// TwinCAT 3 PLC project kittingDeca
// ProgramVersion: 3.1.4023.0
// libraries:
//   Tc2_EtherCAT, * (Beckhoff Automation GmbH)
//   Tc2_MC2, * (Beckhoff Automation GmbH)
//   Tc2_SerialCom, * (Beckhoff Automation GmbH)
//   Tc2_Standard, * (Beckhoff Automation GmbH)
//   Tc2_System, * (Beckhoff Automation GmbH)
//   Tc2_Utilities, * (Beckhoff Automation GmbH)
//   Tc3_Module, * (Beckhoff Automation GmbH)
//   VisuDialogs, * (System)
//   VisuSymbols,3.5.10.0,System
// project tree:
//   DUTs/ user_defined_structure.TcDUT
//   / GlobalTextList.TcGTLO, PlcTask.TcTTO, VISU_TASK.TcTTO, 视图管理器.TcVMO (not stored)
//   GVLs/ E_DOutputMode.TcDUT, E_State.TcDUT, ST_DIO.TcDUT, ST_IO.TcDUT, ST_IO_16.TcDUT, ST_IO_16_int.TcDUT
//   GVLs/kitting deca/axis/ AxisHMI_Ex.TcVIS, E_HomingSteps.TcDUT, FB_MotionAxis_MC.TcPOU, MC_HomeAxis.TcPOU, ST_MotionAxis_MC.TcDUT
//   GVLs/kitting deca/ DigitalInputStatus.TcDUT, FB_DigitalInput.TcPOU, FB_do.TcPOU, FB_PhotoSensor.TcPOU, Roller.TcDUT, Sensor.TcDUT, Valve.TcDUT
//   GVLs/kitting deca/measuring/ ST_byte.TcDUT, ST_IO_byte.TcDUT
//   GVLs/kitting deca/picking module/ Belt.TcDUT, Buffer.TcDUT, Inner_conveyor.TcDUT, PM_others.TcDUT, Outter_coveyor.TcDUT, Picking_Module.TcDUT, RFID.TcDUT
//   GVLs/kitting deca/replenishment module/ arLiftAxis.TcDUT, Infeed.TcDUT, Lift.TcDUT, Outfeed.TcDUT, Replenishment_Module.TcDUT
//   POUs/ E_RemIndex.TcDUT, FB_axisCtrl.TcPOU, FB_remAxisMapping.TcPOU, FB_pmAxisMapping.TcPOU, FB_remIOmapping.TcPOU, FB_rmIOmapping.TcPOU, G_HMI.TcGVL, GVL.TcGVL, G_IO.TcGVL, MAIN.TcPOU, ST_axisCtrl.TcDUT, ST_Color.TcDUT
//   VISUs/ OtherList.TcVIS, visu_PM.TcVIS, visu_ReM.TcVIS, visu_MLC.TcVIS, visu_main.TcVIS, ReMList.TcVIS, PMList.TcVIS, v_byte.TcVIS, v_IO_ReM.TcVIS, v_rem_0.TcVIS, v_pm_0.TcVIS, v_rem_1.TcVIS
// real-time tasks:
//   TASK PlcTask: cycle T#1ms, priority 20, ADS port 350
//   TASK VISU_TASK: cycle T#200000us, priority 30, ADS port 351
// motion (NC):
//   TASK NC-Task 1 SAF: cycle T#2ms, priority 4, ADS port 501
//   TASK NC-Task 1 SVB: cycle T#10ms, priority 8, ADS port 511
//   AXIS rem0_Lift0 (id 4)
//     Dynamic: Acceleration=15000, Deceleration=15000, Jerk=150000
//     Velo: Maximum=3000
//     OtherSettings: AllowMotionCmdToSlave=true
//     encoder EncType=19
//       EncPara: ScaleFactorNumerator=5, ScaleFactorDenominator=262144, Inverse=true, MaxCount=#xffffffff
//         Inc: RefSoftSyncMask=#x00040000
//     drive DrvType=16
//       DrvPara: Inverse=true, MaxCount=#xffffffff, DriveControlDWord=#x00020100
//         Analog: VeloReferenz=500, TorqueSetpointScale=10, ScaleFactorActTorque=0.1
//         TimeComp: TaskDelayCycles=1
//     controller CtrType=1
//       CtrPara: PriorControlFactor=1
//         PosDiffControl: Range=30
//         Observer: BandWidth=20
//   AXIS rem0_Lift1 (id 5)
//     Dynamic: Acceleration=15000, Deceleration=15000, Jerk=150000
//     Velo: Maximum=3000
//     OtherSettings: AllowMotionCmdToSlave=true
//     encoder EncType=19
//       EncPara: ScaleFactorNumerator=5, ScaleFactorDenominator=262144, Inverse=true, MaxCount=#xffffffff
//         Inc: RefSoftSyncMask=#x00040000
//     drive DrvType=16
//       DrvPara: Inverse=true, MaxCount=#xffffffff, DriveControlDWord=#x00020100
//         Analog: VeloReferenz=500, TorqueSetpointScale=10, ScaleFactorActTorque=0.1
//         TimeComp: TaskDelayCycles=1
//     controller CtrType=1
//       CtrPara: PriorControlFactor=1
//         PosDiffControl: Range=30
//         Observer: BandWidth=20
//   AXIS rem1_Lift0 (id 1)
//     Dynamic: Acceleration=15000, Deceleration=15000, Jerk=150000
//     Velo: Maximum=3000
//     OtherSettings: AllowMotionCmdToSlave=true
//     encoder EncType=1
//       EncPara: ScaleFactorNumerator=5, ScaleFactorDenominator=262144, Inverse=true
//         Inc: RefSoftSyncMask=#x00040000
//     drive DrvType=5
//       DrvPara: Inverse=true
//         Analog: VeloReferenz=500, TorqueSetpointScale=10, ScaleFactorActTorque=0.1
//         TimeComp: TaskDelayCycles=1
//     controller CtrType=1
//       CtrPara: PriorControlFactor=1
//         PosDiffControl: Range=30
//         Observer: BandWidth=20
//   AXIS rem1_Lift1 (id 2)
//     Dynamic: Acceleration=15000, Deceleration=15000, Jerk=150000
//     Velo: Maximum=3000
//     OtherSettings: AllowMotionCmdToSlave=true
//     encoder EncType=1
//       EncPara: ScaleFactorNumerator=5, ScaleFactorDenominator=262144, Inverse=true
//         Inc: RefSoftSyncMask=#x00040000
//     drive DrvType=5
//       DrvPara: Inverse=true
//         Analog: VeloReferenz=500, TorqueSetpointScale=10, ScaleFactorActTorque=0.1
//         TimeComp: TaskDelayCycles=1
//     controller CtrType=1
//       CtrPara: PriorControlFactor=1
//         PosDiffControl: Range=30
//         Observer: BandWidth=20
// I/O:
//   DEVICE LB Test (EtherCAT) (disabled), AmsNetId 172.18.236.248.8.1
//     Box 19 (GL20-RTU-ECT) [GL20-RTU-ECT_1.3.5.0]
//       modules: Module 1 (GL20-1600END), Module 2 (GL20-0016ETP)
//     Drive 20 (InoMD800) [MD800_ECAT_9Axis_V0.19]
//   DEVICE ReM test, AmsNetId 192.168.11.159.7.2
//     Box 8 (GL20-RTU-ECT) [GL20-RTU-ECT_1.3.5.0]
//       modules: Module 1 (GL20-1600END), Module 2 (GL20-1600END), Module 3 (GL20-1600END), Module 4 (GL20-1600END), Module 5 (GL20-0016ETP), Module 6 (GL20-0016ETP)
//     rem0_lift0(InoSV630N) [SV630_1Axis_03713]
//     rem0_lift1(InoSV630N) [SV630_1Axis_03713]
//     Box 22 (C2S-EC) [C2S-EC]
//       modules: Module 1 (C2S-EC-24B)
//     Box 25 (6076924) [SIG350-0006AP100] (disabled)
//       modules: Module 1 (IOL_32/32_I/O-Bytes), Module 2 (IOL_32/32_I/O-Bytes), Module 3 (Digital_IN), Module 4 (Digital_IN), Module 5 (Digital_IN), Module 6 (Digital_IN), Module 7 (Digital_IN), Module 8 (Digital_IN)
// variable links:
//   NC-Task 1 SAF/Axes/rem0_Lift0 <-> ReM test/rem0_lift0(InoSV630N)
//     Drive/Inputs/In/nDataIn1 <-> Inputs/Following error actual value
//     Drive/Inputs/In/nDataIn3[0] <-> Inputs/Torque actual value
//     Drive/Inputs/In/nDcOutputTime <-> InfoData/DcOutputShift
//     Drive/Inputs/In/nState1 <-> Inputs/Statusword
//     Drive/Inputs/In/nState2 <-> Inputs/Statusword @bit 8
//     Drive/Inputs/In/nState4 @bit 1 <-> WcState/InputToggle
//     Drive/Inputs/In/nState4 <-> WcState/WcState
//     Drive/Outputs/Out/nCtrl1 <-> Outputs/Controlword
//     Drive/Outputs/Out/nCtrl2 <-> Outputs/Controlword @bit 8
//     Drive/Outputs/Out/nDataOut1 <-> Outputs/Target position
//     Enc/Inputs/In/nDataIn1 <-> Inputs/Position actual value
//     Enc/Inputs/In/nDataIn3 <-> Inputs/Touch probe pos1 pos value
//     Enc/Inputs/In/nDataIn5 <-> Inputs/Touch probe pos2 pos value
//     Enc/Inputs/In/nDcInputTime <-> InfoData/DcInputShift
//     Enc/Inputs/In/nState4 @bit 1 <-> WcState/InputToggle
//     Enc/Inputs/In/nState4 <-> WcState/WcState
//     Enc/Inputs/In/nState5 <-> Inputs/Touch probe status
//     Enc/Inputs/In/nState6 <-> Inputs/Touch probe status @bit 8
//     Enc/Outputs/Out/nCtrl5 <-> Outputs/Touch probe function
//     Enc/Outputs/Out/nCtrl6 <-> Outputs/Touch probe function @bit 8
//   NC-Task 1 SAF/Axes/rem0_Lift1 <-> ReM test/rem0_lift1(InoSV630N)
//     Drive/Inputs/In/nDataIn1 <-> Inputs/Following error actual value
//     Drive/Inputs/In/nDataIn3[0] <-> Inputs/Torque actual value
//     Drive/Inputs/In/nDcOutputTime <-> InfoData/DcOutputShift
//     Drive/Inputs/In/nState1 <-> Inputs/Statusword
//     Drive/Inputs/In/nState2 <-> Inputs/Statusword @bit 8
//     Drive/Inputs/In/nState4 @bit 1 <-> WcState/InputToggle
//     Drive/Inputs/In/nState4 <-> WcState/WcState
//     Drive/Outputs/Out/nCtrl1 <-> Outputs/Controlword
//     Drive/Outputs/Out/nCtrl2 <-> Outputs/Controlword @bit 8
//     Drive/Outputs/Out/nDataOut1 <-> Outputs/Target position
//     Enc/Inputs/In/nDataIn1 <-> Inputs/Position actual value
//     Enc/Inputs/In/nDataIn3 <-> Inputs/Touch probe pos1 pos value
//     Enc/Inputs/In/nDataIn5 <-> Inputs/Touch probe pos2 pos value
//     Enc/Inputs/In/nDcInputTime <-> InfoData/DcInputShift
//     Enc/Inputs/In/nState4 @bit 1 <-> WcState/InputToggle
//     Enc/Inputs/In/nState4 <-> WcState/WcState
//     Enc/Inputs/In/nState5 <-> Inputs/Touch probe status
//     Enc/Inputs/In/nState6 <-> Inputs/Touch probe status @bit 8
//     Enc/Outputs/Out/nCtrl5 <-> Outputs/Touch probe function
//     Enc/Outputs/Out/nCtrl6 <-> Outputs/Touch probe function @bit 8
//   kittingDeca/kittingDeca Instance <-> NC-Task 1 SAF/Axes/rem0_Lift0
//     PlcTask Inputs/GVL.rem[0].lift[0].AxisRef.NcToPlc <-> Outputs/ToPlc
//     PlcTask Outputs/GVL.rem[0].lift[0].AxisRef.PlcToNc <-> Inputs/FromPlc
//   kittingDeca/kittingDeca Instance <-> NC-Task 1 SAF/Axes/rem0_Lift1
//     PlcTask Inputs/GVL.rem[0].lift[1].AxisRef.NcToPlc <-> Outputs/ToPlc
//     PlcTask Outputs/GVL.rem[0].lift[1].AxisRef.PlcToNc <-> Inputs/FromPlc

CONFIGURATION kittingDeca
    RESOURCE PLC ON TwinCAT3
        TASK PlcTask(INTERVAL := T#1ms, PRIORITY := 20);
        TASK VISU_TASK(INTERVAL := T#200000us, PRIORITY := 30);
        PROGRAM MAIN WITH PlcTask : MAIN;
        PROGRAM VisuElems_Visu_Prg WITH VISU_TASK : VisuElems.Visu_Prg;
    END_RESOURCE
END_CONFIGURATION

// ---- DUTs/user_defined_structure.TcDUT
{attribute 'pack_mode' := '1'}
TYPE user_defined_structure :
STRUCT
	a:BOOL;
	b:INT;
	c:STRING;
	d:REAL;
END_STRUCT
END_TYPE

// ---- GVLs/E_DOutputMode.TcDUT
{attribute 'qualified_only'}
{attribute 'strict'}
TYPE E_DOutputMode :
(
	AutoPLC 	:= 0,
	ManualHMI	:= 1
);
END_TYPE

// ---- GVLs/E_State.TcDUT
{attribute 'qualified_only'}
{attribute 'strict'}
TYPE E_State :
(
	DISABLE		:= 0,
	READY 		:= 1,
	WARNING		:= 2,
	ERROR		:= 3
	
);
END_TYPE

// ---- GVLs/kitting deca/axis/E_HomingSteps.TcDUT
TYPE E_HomingSteps :
(
	IDLE 				:= 0,
	INIT				:= 5,
	READ_AND_SAVE_PARAM	:= 10,
	DISABLE_SOFT_LIM	:= 15,
	ENABLE_JOG			:= 20,
	HOMING				:= 25,
	SET_POSITION		:= 30,
	START					:=	40,
	CHECK					:=	45,
	JOG_FW					:=	100,
	JOG_BW_DOG				:=	105,
	FW_DOG_OFF				:=	110,
	BW_DOG_ON				:=	115,
	
	JOG_BW					:=	130,
	JOG_FW_DOG				:=	135,
	BW_DOG_OFF				:=	140,
	FW_DOG_ON				:=	145,
	MCHOME					:=	150,
	WAIT					:=	160,
	DONE				:= 800,
	ERROR				:= 900
);
END_TYPE

// ---- GVLs/kitting deca/axis/ST_MotionAxis_MC.TcDUT
TYPE ST_MotionAxis_MC :
STRUCT
	rVelocity						: 	LREAL   						;
	rVelocity2						: 	LREAL   						;
	rMaxVelocity					:	LREAL							;	
	rAcceleration					:	LREAL							;
	rMaxAcceleration				:	LREAL							;
	rDeceleration					:	LREAL   						;
	rMaxDeceleration				:	LREAL							;
	rJerk							:	LREAL							;
	rMaxJerk						:	LREAL							;
	rPosition						:	LREAL							;
	rSetPosDistance					:	LREAL							;
	rSetPos							: 	LREAL							;	
	rDistance						:   LREAL							;
	rDistance2						:   LREAL							;	
	
	rActualPosSet					:	LREAL							;//ADD BY EVAN 
	rVelocitySet					: 	LREAL   						;//ADD BY EVAN 	
	xHoming							:	BOOL							;//ADD BY EVAN 
	
	rMaxDistance					:	LREAL							;
	bLimit							:   BOOL							;
	bNegLim							:   BOOL							;
	bPosLim							:	BOOL							;
	bNegSen							:   BOOL							;
	bPosSen							:	BOOL							;
	bPositionSensor					:	BOOL							;
	rHomePos						:	LREAL							;
	rActualPos						:	LREAL							;
	PosDiff							:	LREAL							;
	rActualCurr						:	LREAL							;
	axisDirection					:	MC_Direction					;
	
	rVeloPers						: 	LREAL							;
	rAccPers						: 	LREAL							;   
	rDecPers						: 	LREAL							;                                             					
	SetHomePos						: 	LREAL							;
	HomeVelo						: 	LREAL							;
	PosDiffTarget					: 	LREAL							;
	rFirstpos						: 	LREAL							;
	iAxisID							:	INT								;
	xhsHomingStart					: 	BOOL							;
	xHomingDone						: 	BOOL							;
	xForceControlStart				: 	BOOL							;
	xFoceControlDone				:	BOOL							;	
	xMoveABSDone					: 	BOOL							;
	xMoveRelDone					:	BOOL							;
	bInCouple						:	BOOL							;//Flag Axis is coupled 
    xMuteAxisErrorMessages			:	BOOL							;                                         					
	//Visible/Hide HMI interfaces                   					
	bHomeButtonShow					:	BOOL							; 
	bNegSensorShow					:	BOOL							; 
	bPosSensorShow					:	BOOL							;
	bBacklashShow					:	BOOL							;
	bUnitDegShow					:	BOOL							;
    bJerkShow						:	BOOL							; 
	bStopButtonShow					:	BOOL							; 
	   
	
	bMoveAbsHMI						:	BOOL;
	rVelocityHMI 					: 	LREAL;
	rActualPosHMI					:	LREAL							;//ADD BY EVAN
	bMChomingEnable					:	BOOL							;                                         				
	// backlash compensation                        	
	rBacklashvalue					:	LREAL							;
	xbacklashEnable					:	BOOL							;                        		                					
	bdirFW							:	BOOL							;// on hard stop homing , define the direction of rotation
	
	ModOp					 		: 	SINT							;// Axis operation mode (8 )

//	==============================	Beckhoff Tc2_MC2 library(motion)	==================================
	mcPower 						: 	MC_Power					    ;(*	Axis power, enable/disable																			*)
	mcAxisStates					:	MC_AxisStates					;(*	Driver Feedback, curr motor stage 																	*)
	mcHalt							: 	MC_Halt							;(*	Stops an axis with a defined braking ramp															*)
	mcHome							: 	MC_Home							;(*	Axis homing scenario and execution																	*)
	mcJog							: 	MC_Jog							;(*	Axis Joging BW/FW																					*)	
	mcMoveAbsolute					: 	MC_MoveAbsolute					;(*	Axis GoTo Absolute position																			*)	
	mcMoveRelative					: 	MC_MoveRelative					;(*	Axis GoTo Step by SetPos +/- actual position														*)
	mcMoveVelocity					: 	MC_MoveVelocity					;(*	Axis GoTo with constant velocity														*)
	mcReadStatus					: 	MC_ReadStatus					;(*	Read Axis statuses from driver																		*)
	mcReset							: 	MC_Reset						;(*	Reset Driver																						*)
	mcStop							: 	MC_Stop							;(*	Stop Driver																							*)
	mcReadActualPosition			:	MC_ReadActualPosition			;(*	Read the current axis position																		*)
	mcSetpoint						: 	MC_SetPosition					;(*	Sets the current axis position to a parameterizable value											*)
	mcWriteBoolParameter			: 	MC_WriteBoolParameter			;(*	Write bool param to driver																			*)
	mcReadBoolParameter				:	MC_ReadBoolParameter			;(*	Read bool param from driver																			*)
	mcAxisParameter					:   MC_AxisParameter				;(*	Data type is used in conjunction with function blocks for reading and writing of axis parameters	*)
	CoeWrt							:	FB_EcCoESdoWrite;											
	
//	======================================================================================================	

//
	iSdoWrite	:INT; //6:clear encoder
	sNetID : STRING;
	nSlaveAddr	:UINT;
	nSubIndex	: BYTE;
	nIndex	: WORD;
	
	iCoeWrt	: INT;

END_STRUCT
END_TYPE

// ---- GVLs/kitting deca/DigitalInputStatus.TcDUT

{attribute 'qualified_only'}
{attribute 'strict'}
TYPE DigitalInputStatus:
(
        LOW := 0,
        HIGH := 1
);
END_TYPE

// ---- GVLs/kitting deca/measuring/ST_byte.TcDUT
TYPE ST_byte :
STRUCT
	arByte				: ARRAY[1..32] OF ST_IO_byte; 	// struct of digital Imputs for use in program and hmi 
END_STRUCT
END_TYPE

// ---- GVLs/kitting deca/measuring/ST_IO_byte.TcDUT
TYPE ST_IO_byte : // struct of digital IO for use in program and hmi 
STRUCT
	Ch : ARRAY[0..7] OF BOOL ;

END_STRUCT
END_TYPE

// ---- GVLs/kitting deca/picking module/Belt.TcDUT
TYPE Belt :
STRUCT
	cmd	: INT;
	freq	: INT;
END_STRUCT
END_TYPE

// ---- GVLs/kitting deca/picking module/Buffer.TcDUT
TYPE Buffer :
STRUCT
	mcAxis 					: FB_MotionAxis_MC;
	st_mcAxis 				: ST_MotionAxis_MC;
	AxisRef					: AXIS_REF;
	axis_sensor	: BOOL;
	power_axis	: BOOL;
	contractor_axis	: BOOL;
	surfae_slot_0	: BOOL;
	surfae_slot_1	: BOOL;
	surfae_slot_2	: BOOL;
	above_fixture_light_curtain	: BOOL;
	lamp_button	: BOOL;
	button	: BOOL;
	locked	: BOOL;
	magnet	: BOOL;
	magnet_locked	: BOOL;
END_STRUCT
END_TYPE

// ---- GVLs/kitting deca/picking module/Inner_conveyor.TcDUT
TYPE Inner_conveyor :
STRUCT
	belt	: ARRAY[0..2] OF Belt;
	valve	: ARRAY[0..2] OF Valve;
	rfid	: ARRAY[0..1] OF RFID;
END_STRUCT
END_TYPE

// ---- GVLs/kitting deca/picking module/PM_others.TcDUT
TYPE PM_others :
STRUCT
	power_inConv	:BOOL;
	contactor_inConv	: BOOL;
	power_outConv	:BOOL;
	contactor_outConv	: BOOL;	
	measuring_light_curtain_a	: ARRAY[0..16] OF BYTE;
	measuring_light_curtain_b	: ARRAY[0..16] OF BYTE;
END_STRUCT
END_TYPE

// ---- GVLs/kitting deca/picking module/Outter_coveyor.TcDUT
TYPE Outter_coveyor :
STRUCT
	belt	: ARRAY[0..1] OF Belt;
	valve	: ARRAY[0..1] OF Valve;
	photo_sensor	: ARRAY[0..1] OF BOOL;	
END_STRUCT
END_TYPE

// ---- GVLs/kitting deca/picking module/Picking_Module.TcDUT
TYPE Picking_Module :
STRUCT
	buffer : ARRAY[0..1]OF Buffer;	
	inConv : Inner_conveyor;
	outConv : Outter_coveyor;
	power_robot			: BOOL;
	contactor_robot		: BOOL;
	power_inConv		: BOOL;
	contactor_inConv	: BOOL;
	power_outConv		: BOOL;
	contactor_outConv	: BOOL;	
	
END_STRUCT
END_TYPE

// ---- GVLs/kitting deca/picking module/RFID.TcDUT
TYPE RFID :
STRUCT
END_STRUCT
END_TYPE

// ---- GVLs/kitting deca/replenishment module/arLiftAxis.TcDUT
TYPE arLiftAxis :
STRUCT
	lift : ARRAY[0..1] OF FB_remAxisMapping;
END_STRUCT
END_TYPE

// ---- GVLs/kitting deca/replenishment module/Infeed.TcDUT
TYPE Infeed :
STRUCT
	roller : Roller;
	valve_stopper : Valve;
	photo_sensor :ARRAY[0..1]OF FB_PhotoSensor;
END_STRUCT
END_TYPE

// ---- GVLs/kitting deca/replenishment module/Lift.TcDUT
TYPE Lift :
STRUCT
	roller : Roller;
	power_axis	: BOOL;
	contactor_axis : BOOL;	
	mcAxis 					: FB_MotionAxis_MC;
	st_mcAxis 				: ST_MotionAxis_MC;
	AxisRef					: AXIS_REF;
	valve_perturbation : ARRAY [0..3] OF Valve;
	valve_clamp	:Valve;
	photo_sensor :ARRAY[0..1]OF FB_PhotoSensor;
	limit_sensor : ARRAY[0..2]OF BOOL;

END_STRUCT
END_TYPE

// ---- GVLs/kitting deca/replenishment module/Outfeed.TcDUT
TYPE Outfeed :
STRUCT
	roller : Roller;
	photo_sensor :ARRAY[0..1]OF FB_PhotoSensor;
END_STRUCT
END_TYPE

// ---- GVLs/kitting deca/replenishment module/Replenishment_Module.TcDUT
TYPE Replenishment_Module :
STRUCT
	infeed : ARRAY[0..1]OF Infeed;
	outfeed : ARRAY[0..1]OF Outfeed;
	lift : ARRAY[0..1]OF Lift;
END_STRUCT
END_TYPE

// ---- GVLs/kitting deca/Roller.TcDUT
TYPE Roller :
STRUCT
	Power  		: BOOL;
	forward  	: BOOL; 
	backward	: BOOL;
	err 		: BOOL;
END_STRUCT
END_TYPE

// ---- GVLs/kitting deca/Sensor.TcDUT
TYPE Sensor :
STRUCT
	
END_STRUCT
END_TYPE

// ---- GVLs/kitting deca/Valve.TcDUT
TYPE Valve :
STRUCT
	extend 		 : BOOL;
	retract		 : BOOL;
	extended 	 : BOOL;
	retracted 	 : BOOL;	
END_STRUCT
END_TYPE

// ---- GVLs/ST_DIO.TcDUT
TYPE ST_DIO :
STRUCT
	arstDI				: ARRAY[0..DiMouduleMAX] OF ST_IO_16_int; 	// struct of digital Imputs for use in program and hmi 
	arstDO				: ARRAY[0..DOMODULEMAX] OF ST_IO_16_int;	// struct of digital Outputs for use in program and hmi 
	eDOutputMode		: E_DOutputMode 					;	// Switch for change sourse of DO (0 from plc, 1 from HMI)
END_STRUCT
END_TYPE

// ---- GVLs/ST_IO.TcDUT
TYPE ST_IO :
STRUCT
	sName			: STRING		;
	iState			: E_State		;
	xState			: REFERENCE TO BOOL 			;
	xStateHMI		: BOOL 			;
	xInvisible		: BOOL			;
	
END_STRUCT
END_TYPE

// ---- GVLs/ST_IO_16.TcDUT
TYPE ST_IO_16: 
STRUCT
	Ch : ARRAY[0..15] OF BOOL  ; 
END_STRUCT
END_TYPE

// ---- GVLs/ST_IO_16_int.TcDUT
TYPE ST_IO_16_int : // struct of digital IO for use in program and hmi 
STRUCT
	Ch : ARRAY[0..15] OF ST_IO ;

END_STRUCT
END_TYPE

// ---- POUs/E_RemIndex.TcDUT
{attribute 'qualified_only'}
{attribute 'strict'}
TYPE E_RemIndex :
(
	REM0		:= 0,
	REM1 		:= 1,
	REM2		:= 2,
	REM3		:= 3,
	REM4		:= 4,
	REM5 		:= 5,
	REM6		:= 6,
	REM7		:= 7,
	REM8		:= 8,
	REM9 		:= 9
);
END_TYPE

// ---- POUs/ST_axisCtrl.TcDUT
TYPE ST_axisCtrl :
STRUCT
	iStatus	: INT;
	iCmd	: INT;
	iSpeed	: INT;
	rPosition	: LREAL;
	sMsg	: STRING;
END_STRUCT
END_TYPE

// ---- POUs/ST_Color.TcDUT
TYPE ST_Color :
STRUCT
	RED			: DWORD	:= 16#FFFF0000;
	YELLOW		: DWORD	:= 16#FFFFFF00;
	GREEN		: DWORD	:= 16#FF00FF00;
	GREY		: DWORD	:= 16#FFBEBEBE;
	WHITE		: DWORD	:= 16#FFFFFFFF;
	BLACK		: DWORD	:= 16#FF000000;
	BLUE		: DWORD	:= 16#FF0000FF;
END_STRUCT
END_TYPE

// ---- POUs/G_HMI.TcGVL
{attribute 'qualified_only'}
VAR_GLOBAL
	iMainFrame : INT;
	iReM: INT;
	iPM	: INT;
END_VAR

// ---- POUs/GVL.TcGVL
{attribute 'qualified_only'}
VAR_GLOBAL CONSTANT

END_VAR
VAR_GLOBAL

	
	
	rem : ARRAY[0..9] OF Replenishment_Module;
	pm	: ARRAY[0..9] OF Picking_Module;
	pmOthers	:ARRAY[0..4] OF PM_others;
	
	

	
    stByte : REFERENCE TO ST_byte;
	ibyteNum			:ARRAY[1..32] OF  INT ;
	stMeasuringLC : ST_byte;
	byteLC AT%I*:ARRAY [1..32] OF BYTE;
	rfidIn AT%I*:ARRAY [0..31] OF BYTE;
	rfidOut AT%Q*:ARRAY [0..31] OF BYTE;
	arIn	: ARRAY[0..3] OF ST_IO_byte;
	arOut	: ARRAY[0..3] OF ST_IO_byte;
	n: INT;
	
	fb_remIOmapping	: ARRAY[0..9] OF FB_remIOmapping;
	fb_remAxisMapping	: ARRAY[0..19] OF FB_remAxisMapping;
	stAxisCtrl_Lift	: ARRAY[0..19]OF ST_axisCtrl;
	fbAxisCtrl_Lift	: ARRAY [0..19] OF FB_axisCtrl;

	fb_rmIOmapping	: ARRAY[0..4] OF FB_rmIOmapping;
	fb_pmAxisMapping	: ARRAY[0..19] OF FB_pmAxisMapping;
	stAxisCtrl_Buffer	: ARRAY[0..19]OF ST_axisCtrl;
	fbAxisCtrl_Buffer	: ARRAY [0..19] OF FB_axisCtrl;
	

	
END_VAR

// ---- POUs/G_IO.TcGVL
{attribute 'global_init_slot' := '40600'}
VAR_GLOBAL CONSTANT
	{attribute 'global_init_slot'}
	DiMouduleMAX 			:	INT	:=	100;
	{attribute 'global_init_slot'}
	DOMODULEMAX 			:	INT	:=	100;
END_VAR

VAR_GLOBAL
	{attribute 'TcContextName':='PlcTask1'}
	arDI	AT%I*		: ARRAY[0..DiMouduleMAX ] OF ST_IO_16;		//  links to Digital input  Modules 
	{attribute 'TcContextName':='PlcTask1'}
	arDO	AT%Q*		: ARRAY[0..DOMODULEMAX ] OF ST_IO_16;		//  links to Digital output Modules

	iDiMouduleMAX		: INT := 100 							; 		//Number of DI module 
	iDOModuleMax		: INT := 100 							; 		//Number of DO module 


	stDIO				: ST_DIO 							;		// struct DIO for use in plc program
		
	{attribute 'TcContextName':='PlcTask1'}
   	

END_VAR

// ---- POUs/MAIN.TcPOU
PROGRAM MAIN
VAR
	test_bool:BOOL;
	test_int:INT;
	test_real:REAL;
	test_string:STRING;
	test_arr_int:ARRAY[1..10] OF INT;
	test_word:WORD;
	test_arr_bool:ARRAY[1..3] OF BOOL;
	test_structure:user_defined_structure;
	test_arr_string:ARRAY[1..3] OF STRING;
	
	fb_Time : FB_LocalSystemTime;

	byte1 : BYTE;
	string1 :STRING;

	
END_VAR

fb_Time(bEnable := TRUE); 

M_mappingIO();
M_measuringLC();
M_rfid();
runEveryCycle();
M_ReM();

METHOD M_mappingIO 
VAR_INPUT
END_VAR
GVL.fb_remIOmapping[0](iReM:= 0);
GVL.fb_remIOmapping[1](iReM:= 1);
GVL.fb_remIOmapping[2](iReM:= 2);
GVL.fb_remIOmapping[3](iReM:= 3);
GVL.fb_remIOmapping[4](iReM:= 4);
GVL.fb_remIOmapping[5](iReM:= 5);
GVL.fb_remIOmapping[6](iReM:= 6);
GVL.fb_remIOmapping[7](iReM:= 7);
GVL.fb_remIOmapping[8](iReM:= 8);
GVL.fb_remIOmapping[9](iReM:= 9);
GVL.fb_remAxisMapping[0](iReM :=0,iLift:=0,nSlaveAddr:=1002);
GVL.fb_remAxisMapping[1](iReM :=0,iLift:=1,nSlaveAddr:=1003);
GVL.fb_remAxisMapping[2](iReM :=1,iLift:=0,nSlaveAddr:=1006);
GVL.fb_remAxisMapping[3](iReM :=1,iLift:=1,nSlaveAddr:=1007);

GVL.fbAxisCtrl_Lift[0](stAxisCtrl:=GVL.stAxisCtrl_Lift[0],IN_OUT:=GVL.rem[0].lift[0].st_mcAxis);
GVL.fbAxisCtrl_Lift[1](stAxisCtrl:=GVL.stAxisCtrl_Lift[1],IN_OUT:=GVL.rem[0].lift[1].st_mcAxis);
GVL.fbAxisCtrl_Lift[2](stAxisCtrl:=GVL.stAxisCtrl_Lift[2],IN_OUT:=GVL.rem[1].lift[0].st_mcAxis);
GVL.fbAxisCtrl_Lift[3](stAxisCtrl:=GVL.stAxisCtrl_Lift[3],IN_OUT:=GVL.rem[1].lift[1].st_mcAxis);


GVL.fb_rmIOmapping[0](iRm:= 0);
GVL.fb_rmIOmapping[0](iRm:= 1);
GVL.fb_rmIOmapping[0](iRm:= 2);
GVL.fb_rmIOmapping[0](iRm:= 3);
GVL.fb_rmIOmapping[0](iRm:= 4);
GVL.fb_pmAxisMapping[0](iPM :=0,iBuffer:=0,nSlaveAddr:=2002);
GVL.fb_pmAxisMapping[1](iPM :=0,iBuffer:=1,nSlaveAddr:=2003);
GVL.fb_pmAxisMapping[2](iPM :=1,iBuffer:=0,nSlaveAddr:=2006);
GVL.fb_pmAxisMapping[3](iPM :=1,iBuffer:=1,nSlaveAddr:=2007);
GVL.fbAxisCtrl_Buffer[0](stAxisCtrl:=GVL.stAxisCtrl_Buffer[0],IN_OUT:=GVL.pm[0].buffer[0].st_mcAxis);
GVL.fbAxisCtrl_Buffer[1](stAxisCtrl:=GVL.stAxisCtrl_Buffer[1],IN_OUT:=GVL.pm[0].buffer[1].st_mcAxis);
GVL.fbAxisCtrl_Buffer[2](stAxisCtrl:=GVL.stAxisCtrl_Buffer[2],IN_OUT:=GVL.pm[1].buffer[0].st_mcAxis);
GVL.fbAxisCtrl_Buffer[3](stAxisCtrl:=GVL.stAxisCtrl_Buffer[3],IN_OUT:=GVL.pm[1].buffer[1].st_mcAxis);

(*GVL.arrSenDetect[1] := G_IO.arDI[4].Ch[0];
GVL.arrSenDetect[2] := G_IO.arDI[4].Ch[1];
GVL.arrSenDetect[3] := G_IO.arDI[4].Ch[2];
GVL.arrSenDetect[4] := G_IO.arDI[4].Ch[3];
GVL.arrSenDetect[5] := G_IO.arDI[4].Ch[4];*)

(*GVL.rem[0].infeed[0].roller.err						:= G_IO.arDI[0].Ch[0];
GVL.rem[0].infeed[0].valve_stopper.extended  		:= G_IO.arDI[0].Ch[1];
GVL.rem[0].infeed[0].valve_stopper.retracted  		:= G_IO.arDI[0].Ch[2];
GVL.rem[0].infeed[0].photo_sensor[0].set_status(G_IO.arDI[0].Ch[3],10,50);
GVL.rem[0].infeed[0].photo_sensor[1].set_status(G_IO.arDI[0].Ch[4],10,50);
GVL.rem[0].outfeed[0].roller.err					:= G_IO.arDI[0].Ch[5];
GVL.rem[0].outfeed[0].photo_sensor[0].set_status(G_IO.arDI[0].Ch[6],10,50);
GVL.rem[0].outfeed[0].photo_sensor[1].set_status(G_IO.arDI[0].Ch[7],10,50);
GVL.rem[0].lift[0].roller.err						:= G_IO.arDI[0].Ch[8];
GVL.rem[0].lift[0].contactor_axis						:= G_IO.arDI[0].Ch[9];
//GVL.rem[0].lift[0].limit_sensor[0]	:= TRUE;
//GVL.rem[0].lift[0].limit_sensor[1]	:= TRUE;
//GVL.rem[0].lift[0].limit_sensor[2]	:= TRUE;
GVL.rem[0].lift[0].limit_sensor[0]	:= G_IO.arDI[0].Ch[10];
GVL.rem[0].lift[0].limit_sensor[1]	:= G_IO.arDI[0].Ch[11];
GVL.rem[0].lift[0].limit_sensor[2]	:= G_IO.arDI[0].Ch[12];
GVL.rem[0].lift[0].valve_perturbation[0].extended  	:= G_IO.arDI[0].Ch[13];
GVL.rem[0].lift[0].valve_perturbation[0].retracted 	:= G_IO.arDI[0].Ch[14];
GVL.rem[0].lift[0].valve_perturbation[1].extended  	:= G_IO.arDI[0].Ch[15];
GVL.rem[0].lift[0].valve_perturbation[1].retracted 	:= G_IO.arDI[1].Ch[0];
GVL.rem[0].lift[0].valve_perturbation[2].extended  	:= G_IO.arDI[1].Ch[1];
GVL.rem[0].lift[0].valve_perturbation[2].retracted 	:= G_IO.arDI[1].Ch[2];
GVL.rem[0].lift[0].valve_perturbation[3].extended  	:= G_IO.arDI[1].Ch[3];
GVL.rem[0].lift[0].valve_perturbation[3].retracted	:= G_IO.arDI[1].Ch[4];
GVL.rem[0].lift[0].valve_clamp.extended  := G_IO.arDI[1].Ch[5];
GVL.rem[0].lift[0].valve_clamp.retracted  := G_IO.arDI[1].Ch[6];
GVL.rem[0].lift[0].photo_sensor[0].set_status(G_IO.arDI[1].Ch[7],10,50);
GVL.rem[0].lift[0].photo_sensor[1].set_status(G_IO.arDI[1].Ch[8],10,50);

G_IO.arDO[0].Ch[0]	:= GVL.rem[0].infeed[0].roller.Power;
G_IO.arDO[0].Ch[1]	:= GVL.rem[0].infeed[0].roller.forward;
G_IO.arDO[0].Ch[2]	:= GVL.rem[0].infeed[0].roller.backward;
G_IO.arDO[0].Ch[3]	:= GVL.rem[0].outfeed[0].roller.Power;
G_IO.arDO[0].Ch[4]	:= GVL.rem[0].outfeed[0].roller.forward;
G_IO.arDO[0].Ch[5]	:= GVL.rem[0].outfeed[0].roller.backward;
G_IO.arDO[0].Ch[6]	:= GVL.rem[0].lift[0].roller.Power;
G_IO.arDO[0].Ch[7]	:= GVL.rem[0].lift[0].roller.forward;
G_IO.arDO[0].Ch[8]	:= GVL.rem[0].lift[0].roller.backward;
G_IO.arDO[0].Ch[9]	:= GVL.rem[0].lift[0].power_axis;
G_IO.arDO[2].Ch[0]	:= GVL.rem[0].infeed[0].valve_stopper.extend;
G_IO.arDO[2].Ch[1]	:= GVL.rem[0].infeed[0].valve_stopper.retract;
G_IO.arDO[2].Ch[2]	:= GVL.rem[0].lift[0].valve_perturbation[0].extend;
G_IO.arDO[2].Ch[4]	:= GVL.rem[0].lift[0].valve_perturbation[1].extend;
G_IO.arDO[2].Ch[6]	:= GVL.rem[0].lift[0].valve_perturbation[2].extend;
G_IO.arDO[2].Ch[8]	:= GVL.rem[0].lift[0].valve_perturbation[3].extend;
G_IO.arDO[2].Ch[10]	:= GVL.rem[0].lift[0].valve_clamp.extend;
G_IO.arDO[2].Ch[11]	:= GVL.rem[0].lift[0].valve_clamp.retract;



GVL.rem[0].infeed[1].roller.err	:= G_IO.arDI[2].Ch[0];
GVL.rem[0].infeed[1].valve_stopper.extended  := G_IO.arDI[2].Ch[1];
GVL.rem[0].infeed[1].valve_stopper.retracted  := G_IO.arDI[2].Ch[2];
GVL.rem[0].infeed[1].photo_sensor[0].set_status(G_IO.arDI[2].Ch[3],10,50);
GVL.rem[0].infeed[1].photo_sensor[1].set_status(G_IO.arDI[2].Ch[4],10,50);
GVL.rem[0].outfeed[1].roller.err	:= G_IO.arDI[2].Ch[5];
GVL.rem[0].outfeed[1].photo_sensor[0].set_status(G_IO.arDI[2].Ch[6],10,50);
GVL.rem[0].outfeed[1].photo_sensor[1].set_status(G_IO.arDI[2].Ch[7],10,50);
GVL.rem[0].lift[1].roller.err	:= G_IO.arDI[2].Ch[8];
GVL.rem[0].lift[1].contactor_axis	:= G_IO.arDI[2].Ch[9];
//GVL.rem[0].lift[1].limit_sensor[0]	:= TRUE;
//GVL.rem[0].lift[1].limit_sensor[1]	:= TRUE;
//GVL.rem[0].lift[1].limit_sensor[2]	:= TRUE;
GVL.rem[0].lift[1].limit_sensor[0]	:= G_IO.arDI[2].Ch[10];
GVL.rem[0].lift[1].limit_sensor[1]	:= G_IO.arDI[2].Ch[11];
GVL.rem[0].lift[1].limit_sensor[2]	:= G_IO.arDI[2].Ch[12];
GVL.rem[0].lift[1].valve_perturbation[0].extended  := G_IO.arDI[2].Ch[13];
GVL.rem[0].lift[1].valve_perturbation[0].retracted  := G_IO.arDI[2].Ch[14];
GVL.rem[0].lift[1].valve_perturbation[1].extended  := G_IO.arDI[2].Ch[15];
GVL.rem[0].lift[1].valve_perturbation[1].retracted  := G_IO.arDI[3].Ch[0];
GVL.rem[0].lift[1].valve_perturbation[2].extended  := G_IO.arDI[3].Ch[1];
GVL.rem[0].lift[1].valve_perturbation[2].retracted  := G_IO.arDI[3].Ch[2];
GVL.rem[0].lift[1].valve_perturbation[3].extended  := G_IO.arDI[3].Ch[3];
GVL.rem[0].lift[1].valve_perturbation[3].retracted  := G_IO.arDI[3].Ch[4];
GVL.rem[0].lift[1].valve_clamp.extended  := G_IO.arDI[3].Ch[5];
GVL.rem[0].lift[1].valve_clamp.retracted  := G_IO.arDI[3].Ch[6];
GVL.rem[0].lift[1].photo_sensor[0].set_status(G_IO.arDI[3].Ch[7],10,50);
GVL.rem[0].lift[1].photo_sensor[1].set_status(G_IO.arDI[3].Ch[8],10,50);

G_IO.arDO[1].Ch[0]	:= GVL.rem[0].infeed[1].roller.Power;
G_IO.arDO[1].Ch[1]	:= GVL.rem[0].infeed[1].roller.forward;
G_IO.arDO[1].Ch[2]	:= GVL.rem[0].infeed[1].roller.backward;
G_IO.arDO[1].Ch[3]	:= GVL.rem[0].outfeed[1].roller.Power;
G_IO.arDO[1].Ch[4]	:= GVL.rem[0].outfeed[1].roller.forward;
G_IO.arDO[1].Ch[5]	:= GVL.rem[0].outfeed[1].roller.backward;
G_IO.arDO[1].Ch[6]	:= GVL.rem[0].lift[1].roller.Power;
G_IO.arDO[1].Ch[7]	:= GVL.rem[0].lift[1].roller.forward;
G_IO.arDO[1].Ch[8]	:= GVL.rem[0].lift[1].roller.backward;
G_IO.arDO[1].Ch[9]	:= GVL.rem[0].lift[1].power_axis;
G_IO.arDO[2].Ch[12]	:= GVL.rem[0].infeed[1].valve_stopper.extend;
G_IO.arDO[2].Ch[13]	:= GVL.rem[0].infeed[1].valve_stopper.retract;
G_IO.arDO[2].Ch[14]	:= GVL.rem[0].lift[1].valve_perturbation[0].extend;
G_IO.arDO[3].Ch[0]	:= GVL.rem[0].lift[1].valve_perturbation[1].extend;
G_IO.arDO[3].Ch[2]	:= GVL.rem[0].lift[1].valve_perturbation[2].extend;
G_IO.arDO[3].Ch[4]	:= GVL.rem[0].lift[1].valve_perturbation[3].extend;
G_IO.arDO[3].Ch[6]	:= GVL.rem[0].lift[1].valve_clamp.extend;
G_IO.arDO[3].Ch[7]	:= GVL.rem[0].lift[1].valve_clamp.retract;*)


//////////////////////////////PM[0]///////////////////////////////////
(*GVL.pm[0].buffer[0].contractor_axis				:= G_IO.arDI[50].Ch[0];
GVL.pm[0].buffer[0].axis_sensor					:= G_IO.arDI[50].Ch[1];
GVL.pm[0].buffer[0].surfae_slot_0				:= G_IO.arDI[50].Ch[2];
GVL.pm[0].buffer[0].surfae_slot_1				:= G_IO.arDI[50].Ch[3];
GVL.pm[0].buffer[0].surfae_slot_2				:= G_IO.arDI[50].Ch[4];
GVL.pm[0].buffer[0].above_fixture_light_curtain	:= G_IO.arDI[50].Ch[5];
GVL.pm[0].buffer[0].button						:= G_IO.arDI[50].Ch[6];
GVL.pm[0].buffer[0].locked						:= G_IO.arDI[50].Ch[7];
GVL.pm[0].buffer[0].magnet_locked				:= G_IO.arDI[50].Ch[8];
GVL.pm[0].buffer[1].contractor_axis				:= G_IO.arDI[50].Ch[9];
GVL.pm[0].buffer[1].axis_sensor					:= G_IO.arDI[50].Ch[10];
GVL.pm[0].buffer[1].surfae_slot_0				:= G_IO.arDI[50].Ch[11];
GVL.pm[0].buffer[1].surfae_slot_1				:= G_IO.arDI[50].Ch[12];
GVL.pm[0].buffer[1].surfae_slot_2				:= G_IO.arDI[50].Ch[13];
GVL.pm[0].buffer[1].above_fixture_light_curtain	:= G_IO.arDI[50].Ch[14];
GVL.pm[0].buffer[1].button						:= G_IO.arDI[50].Ch[15];
GVL.pm[0].buffer[1].locked						:= G_IO.arDI[51].Ch[0];
GVL.pm[0].buffer[1].magnet_locked				:= G_IO.arDI[51].Ch[1];
GVL.pm[0].contactor_robot						:= G_IO.arDI[51].Ch[2];
GVL.pm[0].inConv.valve[0].extended				:= G_IO.arDI[51].Ch[3];
GVL.pm[0].inConv.valve[0].retracted				:= G_IO.arDI[51].Ch[4];
GVL.pm[0].inConv.valve[1].extended				:= G_IO.arDI[51].Ch[5];
GVL.pm[0].inConv.valve[1].retracted				:= G_IO.arDI[51].Ch[6];
GVL.pm[0].inConv.valve[2].extended				:= G_IO.arDI[51].Ch[7];
GVL.pm[0].inConv.valve[2].retracted				:= G_IO.arDI[51].Ch[8];
GVL.pm[0].outConv.photo_sensor[0]				:= G_IO.arDI[51].Ch[9];
GVL.pm[0].outConv.photo_sensor[1]				:= G_IO.arDI[51].Ch[10];
GVL.pm[0].outConv.valve[0].extended				:= G_IO.arDI[51].Ch[11];
GVL.pm[0].outConv.valve[0].retracted			:= G_IO.arDI[51].Ch[12];
GVL.pm[0].outConv.valve[1].extended				:= G_IO.arDI[51].Ch[13];
GVL.pm[0].outConv.valve[1].retracted			:= G_IO.arDI[51].Ch[14];


GVL.pm[0].contactor_inConv						:= G_IO.arDI[54].Ch[0];//share with pm[1]
GVL.pm[0].contactor_inConv						:= G_IO.arDI[54].Ch[1];//share with pm[1]

G_IO.arDO[50].Ch[0]	:= GVL.pm[0].buffer[0].power_axis;
G_IO.arDO[50].Ch[1]	:= GVL.pm[0].buffer[0].magnet;
G_IO.arDO[50].Ch[2]	:= GVL.pm[0].buffer[1].power_axis;
G_IO.arDO[50].Ch[3]	:= GVL.pm[0].buffer[1].magnet;
G_IO.arDO[50].Ch[4]	:= GVL.pm[0].power_robot;
G_IO.arDO[50].Ch[12]	:= GVL.pm[0].buffer[0].lamp_button;
G_IO.arDO[50].Ch[13]	:= GVL.pm[0].buffer[1].lamp_button;

G_IO.arDO[52].Ch[0]	:= GVL.pm[0].inConv.valve[0].extend;
G_IO.arDO[52].Ch[2]	:= GVL.pm[0].inConv.valve[1].extend;
G_IO.arDO[52].Ch[4]	:= GVL.pm[0].inConv.valve[2].extend;
G_IO.arDO[52].Ch[6]	:= GVL.pm[0].outConv.valve[0].extend;
G_IO.arDO[52].Ch[8]	:= GVL.pm[0].outConv.valve[1].extend;

G_IO.arDO[50].Ch[10]	:= GVL.pm[0].power_inConv;//share with pm[1]
G_IO.arDO[50].Ch[11]	:= GVL.pm[0].power_outConv;//share with pm[1]
*)
END_METHOD

METHOD M_measuringLC : BOOL
VAR_INPUT
END_VAR

VAR
	i: INT;
	j: INT;
END_VAR
FOR i :=1 TO 32 DO
	GVL.ibyteNum[i] := i;
END_FOR
FOR i:=1 TO 32 DO	
	GVL.stMeasuringLC.arByte[i].Ch[0]	:= GVL.byteLC[i].0;
	GVL.stMeasuringLC.arByte[i].Ch[1]	:= GVL.byteLC[i].1;
	GVL.stMeasuringLC.arByte[i].Ch[2]	:= GVL.byteLC[i].2;
	GVL.stMeasuringLC.arByte[i].Ch[3]	:= GVL.byteLC[i].3;
	GVL.stMeasuringLC.arByte[i].Ch[4]	:= GVL.byteLC[i].4;
	GVL.stMeasuringLC.arByte[i].Ch[5]	:= GVL.byteLC[i].5;
	GVL.stMeasuringLC.arByte[i].Ch[6]	:= GVL.byteLC[i].6;
	GVL.stMeasuringLC.arByte[i].Ch[7]	:= GVL.byteLC[i].7;
END_FOR


GVL.stByte REF= GVL.stMeasuringLC;
END_METHOD

METHOD M_ReM : BOOL
VAR_INPUT
END_VAR

//========== Lift0 Axis Config ==========
(*GVL.rem[0].lift[0].mcAxis
(
	ZSN		:= GVL.rem[0].lift[0].limit_sensor[2] OR GVL.rem[0].lift[0].st_mcAxis.xHoming,
	ZSP		:= GVL.rem[0].lift[0].limit_sensor[1]	OR GVL.rem[0].lift[0].st_mcAxis.xHoming,
	IN_OUT	:= GVL.rem[0].lift[0].st_mcAxis, 
	AXIS	:= GVL.rem[0].lift[0].Axisref, 
);
GVL.rem[0].lift[0].st_mcAxis.bPosSensorShow	:= TRUE;
GVL.rem[0].lift[0].st_mcAxis.bNegSensorShow	:= TRUE;
GVL.rem[0].lift[0].st_mcAxis.bStopButtonShow	:= TRUE;
GVL.rem[0].lift[0].st_mcAxis.rMaxAcceleration	:= 50000;
GVL.rem[0].lift[0].st_mcAxis.rMaxDeceleration	:= 50000;
GVL.rem[0].lift[0].st_mcAxis.rMaxJerk			:= 500000;
GVL.rem[0].lift[0].st_mcAxis.rAcceleration	:= 2500;
GVL.rem[0].lift[0].st_mcAxis.rDeceleration	:= 2500;
GVL.rem[0].lift[0].st_mcAxis.rJerk			:= 12500;
GVL.rem[0].lift[0].st_mcAxis.rMaxVelocity		:= 100;
GVL.rem[0].lift[0].st_mcAxis.rMaxDistance		:= 50;
GVL.rem[0].lift[0].st_mcAxis.bPosSen	:= GVL.rem[0].lift[0].limit_sensor[1] ;
GVL.rem[0].lift[0].st_mcAxis.bNegSen	:= GVL.rem[0].lift[0].limit_sensor[2] ;
GVL.rem[0].lift[0].st_mcAxis.mcHome.bCalibrationCam	:= GVL.rem[0].lift[0].limit_sensor[0];
GVL.rem[0].lift[0].st_mcAxis.bPositionSensor	:= GVL.rem[0].lift[0].limit_sensor[0];
GVL.rem[0].lift[0].st_mcAxis.bdirFW	:= TRUE;
GVL.rem[0].lift[0].st_mcAxis.rSetPos	:= 0;
GVL.rem[0].lift[0].st_mcAxis.sNetID := '192.168.11.159.1.1';
GVL.rem[0].lift[0].st_mcAxis.nSlaveAddr	:= 1002;
//GVL.rem[0].lift[0].st_mcAxis.nSubIndex := 16#1F;
//GVL.rem[0].lift[0].st_mcAxis.nIndex	:= 16#2005;


//========== Lift1 Axis Config ==========
GVL.rem[0].lift[1].mcAxis
(
	ZSN		:= GVL.rem[0].lift[1].limit_sensor[2] OR GVL.rem[0].lift[1].st_mcAxis.xHoming,
	ZSP		:= GVL.rem[0].lift[1].limit_sensor[1]	OR GVL.rem[0].lift[1].st_mcAxis.xHoming,
	IN_OUT	:= GVL.rem[0].lift[1].st_mcAxis, 
	AXIS	:= GVL.rem[0].lift[1].Axisref, 
);
GVL.rem[0].lift[1].st_mcAxis.bPosSensorShow	:= TRUE;
GVL.rem[0].lift[1].st_mcAxis.bNegSensorShow	:= TRUE;
GVL.rem[0].lift[1].st_mcAxis.bStopButtonShow	:= TRUE;
GVL.rem[0].lift[1].st_mcAxis.rMaxAcceleration	:= 50000;
GVL.rem[0].lift[1].st_mcAxis.rMaxDeceleration	:= 50000;
GVL.rem[0].lift[1].st_mcAxis.rMaxJerk			:= 500000;
GVL.rem[0].lift[1].st_mcAxis.rAcceleration	:= 2500;
GVL.rem[0].lift[1].st_mcAxis.rDeceleration	:= 2500;
GVL.rem[0].lift[1].st_mcAxis.rJerk			:= 12500;
GVL.rem[0].lift[1].st_mcAxis.rMaxVelocity		:= 100;
GVL.rem[0].lift[1].st_mcAxis.rMaxDistance		:= 50;
GVL.rem[0].lift[1].st_mcAxis.bPosSen	:= GVL.rem[0].lift[1].limit_sensor[1] ;
GVL.rem[0].lift[1].st_mcAxis.bNegSen	:= GVL.rem[0].lift[1].limit_sensor[2] ;
GVL.rem[0].lift[1].st_mcAxis.mcHome.bCalibrationCam	:= GVL.rem[0].lift[1].limit_sensor[0];
GVL.rem[0].lift[1].st_mcAxis.bPositionSensor	:= GVL.rem[0].lift[1].limit_sensor[0];
GVL.rem[0].lift[1].st_mcAxis.bdirFW	:= TRUE;
GVL.rem[0].lift[1].st_mcAxis.rSetPos	:= 0;
GVL.rem[0].lift[1].st_mcAxis.sNetID := '192.168.11.159.1.1';
GVL.rem[0].lift[1].st_mcAxis.nSlaveAddr	:= 1003;
//GVL.rem[0].lift[1].st_mcAxis.nSubIndex := 16#1F;
//GVL.rem[0].lift[1].st_mcAxis.nIndex	:=  16#2005;

CASE GVL.iFRtest OF 
	0:		
		//IF GVL.rem[0].lift[0].st_mcAxis.xHomingDone THEN
			IF GVL.bTs1 THEN
				GVL.rem[0].lift[0].st_mcAxis.mcMoveAbsolute.Execute := FALSE;
				GVL.iFRtest :=1;
			END_IF
		//END_IF
	1://open positon
		GVL.rem[0].lift[0].st_mcAxis.rActualPosSet := 0;
		GVL.rem[0].lift[0].st_mcAxis.rVelocitySet := 300;			
		GVL.rem[0].lift[0].st_mcAxis.mcMoveAbsolute.Execute := TRUE;
		GVL.rem[0].lift[1].st_mcAxis.rActualPosSet := 0;
		GVL.rem[0].lift[1].st_mcAxis.rVelocitySet := 300;			
		GVL.rem[0].lift[1].st_mcAxis.mcMoveAbsolute.Execute := TRUE;
		IF GVL.rem[0].lift[0].st_mcAxis.mcMoveAbsolute.Done AND GVL.rem[0].lift[1].st_mcAxis.mcMoveAbsolute.Done THEN
			GVL.rem[0].lift[0].st_mcAxis.mcMoveAbsolute.Execute := FALSE;
			GVL.rem[0].lift[1].st_mcAxis.mcMoveAbsolute.Execute := FALSE;
			GVL.iFRtest := 2;
		END_IF
	
	2:
		ton_delay.IN := TRUE;
		IF ton_delay.Q THEN
			ton_delay.IN := FALSE;
			GVL.iFRtest := 3;
		END_IF
	3://close position
		GVL.rem[0].lift[0].st_mcAxis.rActualPosSet := 424;
		GVL.rem[0].lift[0].st_mcAxis.rVelocitySet := 300;			
		GVL.rem[0].lift[0].st_mcAxis.mcMoveAbsolute.Execute := TRUE;
		GVL.rem[0].lift[1].st_mcAxis.rActualPosSet := 424;
		GVL.rem[0].lift[1].st_mcAxis.rVelocitySet := 300;			
		GVL.rem[0].lift[1].st_mcAxis.mcMoveAbsolute.Execute := TRUE;		
		GVL.st_mcAxis[1].mcMoveAbsolute.Execute := TRUE;
			IF GVL.rem[0].lift[0].st_mcAxis.mcMoveAbsolute.Done AND GVL.rem[0].lift[1].st_mcAxis.mcMoveAbsolute.Done THEN
				GVL.rem[0].lift[0].st_mcAxis.mcMoveAbsolute.Execute := FALSE;
				GVL.rem[0].lift[1].st_mcAxis.mcMoveAbsolute.Execute := FALSE;
				GVL.iFRtest := 4;
			END_IF   
	4://delay
		ton_delay.IN := TRUE;
		IF ton_delay.Q THEN
			ton_delay.IN := FALSE;
			GVL.iFRtest := 5;
		END_IF
	5://open positon
		GVL.rem[0].lift[0].st_mcAxis.rActualPosSet := 0;
		GVL.rem[0].lift[0].st_mcAxis.rVelocitySet := 300;			
		GVL.rem[0].lift[0].st_mcAxis.mcMoveAbsolute.Execute := TRUE;
		GVL.rem[0].lift[1].st_mcAxis.rActualPosSet := 0;
		GVL.rem[0].lift[1].st_mcAxis.rVelocitySet := 300;			
		GVL.rem[0].lift[1].st_mcAxis.mcMoveAbsolute.Execute := TRUE;
		IF GVL.rem[0].lift[0].st_mcAxis.mcMoveAbsolute.Done AND GVL.rem[0].lift[1].st_mcAxis.mcMoveAbsolute.Done THEN
			GVL.rem[0].lift[0].st_mcAxis.mcMoveAbsolute.Execute := FALSE;
			GVL.rem[0].lift[1].st_mcAxis.mcMoveAbsolute.Execute := FALSE;
			GVL.iFRtest := 6;
		END_IF
	6:
		GVL.iFRtest := 0;
END_CASE*)
END_METHOD

METHOD M_rfid : BOOL
VAR_INPUT
END_VAR

VAR
	i: INT;
	
END_VAR
byte1 := ASC(string1);
FOR i:=0 TO 3 DO	
	GVL.arIn[i].Ch[0]	:= GVL.rfidIn[i].0;
	GVL.arIn[i].Ch[1]	:= GVL.rfidIn[i].1;
	GVL.arIn[i].Ch[2]	:= GVL.rfidIn[i].2;
	GVL.arIn[i].Ch[3]	:= GVL.rfidIn[i].3;
	GVL.arIn[i].Ch[4]	:= GVL.rfidIn[i].4;
	GVL.arIn[i].Ch[5]	:= GVL.rfidIn[i].5;
	GVL.arIn[i].Ch[6]	:= GVL.rfidIn[i].6;
	GVL.arIn[i].Ch[7]	:= GVL.rfidIn[i].7;
	GVL.rfidOut[i].0	:= GVL.arOut[i].Ch[0];
	GVL.rfidOut[i].1	:= GVL.arOut[i].Ch[1];
	GVL.rfidOut[i].2	:= GVL.arOut[i].Ch[2];
	GVL.rfidOut[i].3	:= GVL.arOut[i].Ch[3];
	GVL.rfidOut[i].4	:= GVL.arOut[i].Ch[4];
	GVL.rfidOut[i].5	:= GVL.arOut[i].Ch[5];
	GVL.rfidOut[i].6	:= GVL.arOut[i].Ch[6];
	GVL.rfidOut[i].7	:= GVL.arOut[i].Ch[7];	
END_FOR

FOR i:=4 TO 31 DO
	GVL.rfidOut[i] := INT_TO_BYTE(28*GVL.n+i-3);
END_FOR
END_METHOD

METHOD runEveryCycle : BOOL
VAR_INPUT
END_VAR

VAR
	


END_VAR
(*
CASE GVL.iFRtest OF 
	0:		
		IF GVL.st_mcAxis[0].xHomingDone THEN
			IF GVL.bTs1 THEN
				GVL.st_mcAxis[0].mcMoveAbsolute.Execute := FALSE;
				GVL.iFRtest :=1;
			END_IF
		END_IF
		IF GVL.bBeltTs THEN
			G_IO.arDI[5].Ch[2] := TRUE;
			G_IO.arDI[5].Ch[3] := TRUE;
			GVL.st_mcAxis[0].mcMoveAbsolute.Execute := FALSE;
			GVL.iFRtest :=100;
		END_IF
	100:
		GVL.st_mcAxis[0].rActualPosSet := 60000000;
		GVL.st_mcAxis[0].rVelocitySet := 150;	
		GVL.st_mcAxis[0].mcMoveAbsolute.Execute := TRUE;	
		IF NOT GVL.bBeltTs THEN
			GVL.st_mcAxis[0].mcMoveAbsolute.Execute := FALSE;
			GVL.st_mcAxis[0].mcStop.Execute := TRUE;
			IF GVL.st_mcAxis[0].mcStop.Done THEN
				GVL.st_mcAxis[0].mcStop.Execute := FALSE;
				GVL.iFRtest :=0;
			END_IF
			
		END_IF
	1://open positon
		valve := FALSE;
		IF retracted THEN
			GVL.st_mcAxis[0].rActualPosSet := 102.8;
			GVL.st_mcAxis[0].rVelocitySet := 300;			
			GVL.st_mcAxis[0].mcMoveAbsolute.Execute := TRUE;
			IF GVL.st_mcAxis[0].mcMoveAbsolute.Done THEN
				GVL.st_mcAxis[0].mcMoveAbsolute.Execute := FALSE;
				GVL.iFRtest := 2;
			END_IF
		END_IF
	2://valve extend
		valve := TRUE;
		IF extended THEN
			GVL.iFRtest := 3;
		END_IF
	3://delay
		ton_delay.IN := TRUE;
		IF ton_delay.Q THEN
			ton_delay.IN := FALSE;
			GVL.iFRtest := 4;
		END_IF
	4://close position
		GVL.st_mcAxis[0].rActualPosSet := -78.4;
		GVL.st_mcAxis[0].rVelocitySet := 300;			
		GVL.st_mcAxis[0].mcMoveAbsolute.Execute := TRUE;
		IF GVL.st_mcAxis[0].mcMoveAbsolute.Done THEN
			GVL.st_mcAxis[0].mcMoveAbsolute.Execute := FALSE;
			GVL.iFRtest := 6;
		END_IF	   
	5://delay
		ton_delay.IN := TRUE;
		IF ton_delay.Q THEN
			ton_delay.IN := FALSE;
			GVL.iFRtest := 6;
		END_IF
	6://valve retract
		valve := FALSE;
		IF retracted THEN
			GVL.iFRtest := 7;
		END_IF	
	7://valve extend
		valve := TRUE;
		IF extended THEN
			GVL.iFRtest := 8;
		END_IF	
	8://delay
		ton_delay.IN := TRUE;
		IF ton_delay.Q THEN
			ton_delay.IN := FALSE;
			GVL.iFRtest := 9;
		END_IF
	9://open positon
		GVL.st_mcAxis[0].rActualPosSet := 102.8;
		GVL.st_mcAxis[0].rVelocitySet := 300;			
		GVL.st_mcAxis[0].mcMoveAbsolute.Execute := TRUE;
		IF GVL.st_mcAxis[0].mcMoveAbsolute.Done THEN
			GVL.st_mcAxis[0].mcMoveAbsolute.Execute := FALSE;
			GVL.iFRtest := 10;
		END_IF
	10:
		GVL.iFRtest := 0;
END_CASE
*)
END_METHOD

END_PROGRAM

// ---- POUs/FB_remIOmapping.TcPOU
FUNCTION_BLOCK FB_remIOmapping
VAR_INPUT
	iReM	: INT;
END_VAR
VAR_OUTPUT
END_VAR
	
VAR
	
END_VAR



GVL.rem[iReM].infeed[0].roller.err						:= G_IO.arDI[iReM*4].Ch[0];
GVL.rem[iReM].infeed[0].valve_stopper.extended  		:= G_IO.arDI[iReM*4].Ch[1];
GVL.rem[iReM].infeed[0].valve_stopper.retracted  		:= G_IO.arDI[iReM*4].Ch[2];
GVL.rem[iReM].infeed[0].photo_sensor[0].set_status(G_IO.arDI[iReM*4].Ch[3],10,50);
GVL.rem[iReM].infeed[0].photo_sensor[1].set_status(G_IO.arDI[iReM*4].Ch[4],10,50);
GVL.rem[iReM].outfeed[0].roller.err					:= G_IO.arDI[iReM*4].Ch[5];
GVL.rem[iReM].outfeed[0].photo_sensor[0].set_status(G_IO.arDI[iReM*4].Ch[6],10,50);
GVL.rem[iReM].outfeed[0].photo_sensor[1].set_status(G_IO.arDI[iReM*4].Ch[7],10,50);
GVL.rem[iReM].lift[0].roller.err						:= G_IO.arDI[iReM*4].Ch[8];
GVL.rem[iReM].lift[0].contactor_axis						:= G_IO.arDI[iReM*4].Ch[9];
//GVL.rem[iReM].lift[0].limit_sensor[0]	:= TRUE;
//GVL.rem[iReM].lift[0].limit_sensor[1]	:= TRUE;
//GVL.rem[iReM].lift[0].limit_sensor[2]	:= TRUE;
GVL.rem[iReM].lift[0].limit_sensor[0]	:= G_IO.arDI[iReM*4].Ch[10];
GVL.rem[iReM].lift[0].limit_sensor[1]	:= G_IO.arDI[iReM*4].Ch[11];
GVL.rem[iReM].lift[0].limit_sensor[2]	:= G_IO.arDI[iReM*4].Ch[12];
GVL.rem[iReM].lift[0].valve_perturbation[0].extended  	:= G_IO.arDI[iReM*4].Ch[13];
GVL.rem[iReM].lift[0].valve_perturbation[0].retracted 	:= G_IO.arDI[iReM*4].Ch[14];
GVL.rem[iReM].lift[0].valve_perturbation[1].extended  	:= G_IO.arDI[iReM*4].Ch[15];
GVL.rem[iReM].lift[0].valve_perturbation[1].retracted 	:= G_IO.arDI[iReM*4+1].Ch[0];
GVL.rem[iReM].lift[0].valve_perturbation[2].extended  	:= G_IO.arDI[iReM*4+1].Ch[1];
GVL.rem[iReM].lift[0].valve_perturbation[2].retracted 	:= G_IO.arDI[iReM*4+1].Ch[2];
GVL.rem[iReM].lift[0].valve_perturbation[3].extended  	:= G_IO.arDI[iReM*4+1].Ch[3];
GVL.rem[iReM].lift[0].valve_perturbation[3].retracted	:= G_IO.arDI[iReM*4+1].Ch[4];
GVL.rem[iReM].lift[0].valve_clamp.extended  := G_IO.arDI[iReM*4+1].Ch[5];
GVL.rem[iReM].lift[0].valve_clamp.retracted  := G_IO.arDI[iReM*4+1].Ch[6];
GVL.rem[iReM].lift[0].photo_sensor[0].set_status(G_IO.arDI[iReM*4+1].Ch[7],10,50);
GVL.rem[iReM].lift[0].photo_sensor[1].set_status(G_IO.arDI[iReM*4+1].Ch[8],10,50);

G_IO.arDO[iReM*4].Ch[0]	:= GVL.rem[iReM].infeed[0].roller.Power;
G_IO.arDO[iReM*4].Ch[1]	:= GVL.rem[iReM].infeed[0].roller.forward;
G_IO.arDO[iReM*4].Ch[2]	:= GVL.rem[iReM].infeed[0].roller.backward;
G_IO.arDO[iReM*4].Ch[3]	:= GVL.rem[iReM].outfeed[0].roller.Power;
G_IO.arDO[iReM*4].Ch[4]	:= GVL.rem[iReM].outfeed[0].roller.forward;
G_IO.arDO[iReM*4].Ch[5]	:= GVL.rem[iReM].outfeed[0].roller.backward;
G_IO.arDO[iReM*4].Ch[6]	:= GVL.rem[iReM].lift[0].roller.Power;
G_IO.arDO[iReM*4].Ch[7]	:= GVL.rem[iReM].lift[0].roller.forward;
G_IO.arDO[iReM*4].Ch[8]	:= GVL.rem[iReM].lift[0].roller.backward;
G_IO.arDO[iReM*4].Ch[9]	:= GVL.rem[iReM].lift[0].power_axis;
G_IO.arDO[iReM*4+2].Ch[0]	:= GVL.rem[iReM].infeed[0].valve_stopper.extend;
G_IO.arDO[iReM*4+2].Ch[1]	:= GVL.rem[iReM].infeed[0].valve_stopper.retract;
G_IO.arDO[iReM*4+2].Ch[2]	:= GVL.rem[iReM].lift[0].valve_perturbation[0].extend;
G_IO.arDO[iReM*4+2].Ch[4]	:= GVL.rem[iReM].lift[0].valve_perturbation[1].extend;
G_IO.arDO[iReM*4+2].Ch[6]	:= GVL.rem[iReM].lift[0].valve_perturbation[2].extend;
G_IO.arDO[iReM*4+2].Ch[8]	:= GVL.rem[iReM].lift[0].valve_perturbation[3].extend;
G_IO.arDO[iReM*4+2].Ch[10]	:= GVL.rem[iReM].lift[0].valve_clamp.extend;
G_IO.arDO[iReM*4+2].Ch[11]	:= GVL.rem[iReM].lift[0].valve_clamp.retract;



GVL.rem[iReM].infeed[1].roller.err	:= G_IO.arDI[iReM*4+2].Ch[0];
GVL.rem[iReM].infeed[1].valve_stopper.extended  := G_IO.arDI[iReM*4+2].Ch[1];
GVL.rem[iReM].infeed[1].valve_stopper.retracted  := G_IO.arDI[iReM*4+2].Ch[2];
GVL.rem[iReM].infeed[1].photo_sensor[0].set_status(G_IO.arDI[iReM*4+2].Ch[3],10,50);
GVL.rem[iReM].infeed[1].photo_sensor[1].set_status(G_IO.arDI[iReM*4+2].Ch[4],10,50);
GVL.rem[iReM].outfeed[1].roller.err	:= G_IO.arDI[iReM*4+2].Ch[5];
GVL.rem[iReM].outfeed[1].photo_sensor[0].set_status(G_IO.arDI[iReM*4+2].Ch[6],10,50);
GVL.rem[iReM].outfeed[1].photo_sensor[1].set_status(G_IO.arDI[iReM*4+2].Ch[7],10,50);
GVL.rem[iReM].lift[1].roller.err	:= G_IO.arDI[iReM*4+2].Ch[8];
GVL.rem[iReM].lift[1].contactor_axis	:= G_IO.arDI[iReM*4+2].Ch[9];
//GVL.rem[iReM].lift[1].limit_sensor[0]	:= TRUE;
//GVL.rem[iReM].lift[1].limit_sensor[1]	:= TRUE;
//GVL.rem[iReM].lift[1].limit_sensor[2]	:= TRUE;
GVL.rem[iReM].lift[1].limit_sensor[0]	:= G_IO.arDI[iReM*4+2].Ch[10];
GVL.rem[iReM].lift[1].limit_sensor[1]	:= G_IO.arDI[iReM*4+2].Ch[11];
GVL.rem[iReM].lift[1].limit_sensor[2]	:= G_IO.arDI[iReM*4+2].Ch[12];
GVL.rem[iReM].lift[1].valve_perturbation[0].extended  := G_IO.arDI[iReM*4+2].Ch[13];
GVL.rem[iReM].lift[1].valve_perturbation[0].retracted  := G_IO.arDI[iReM*4+2].Ch[14];
GVL.rem[iReM].lift[1].valve_perturbation[1].extended  := G_IO.arDI[iReM*4+2].Ch[15];
GVL.rem[iReM].lift[1].valve_perturbation[1].retracted  := G_IO.arDI[iReM*4+3].Ch[0];
GVL.rem[iReM].lift[1].valve_perturbation[2].extended  := G_IO.arDI[iReM*4+3].Ch[1];
GVL.rem[iReM].lift[1].valve_perturbation[2].retracted  := G_IO.arDI[iReM*4+3].Ch[2];
GVL.rem[iReM].lift[1].valve_perturbation[3].extended  := G_IO.arDI[iReM*4+3].Ch[3];
GVL.rem[iReM].lift[1].valve_perturbation[3].retracted  := G_IO.arDI[iReM*4+3].Ch[4];
GVL.rem[iReM].lift[1].valve_clamp.extended  := G_IO.arDI[iReM*4+3].Ch[5];
GVL.rem[iReM].lift[1].valve_clamp.retracted  := G_IO.arDI[iReM*4+3].Ch[6];
GVL.rem[iReM].lift[1].photo_sensor[0].set_status(G_IO.arDI[iReM*4+3].Ch[7],10,50);
GVL.rem[iReM].lift[1].photo_sensor[1].set_status(G_IO.arDI[iReM*4+3].Ch[8],10,50);

G_IO.arDO[iReM*4+1].Ch[0]	:= GVL.rem[iReM].infeed[1].roller.Power;
G_IO.arDO[iReM*4+1].Ch[1]	:= GVL.rem[iReM].infeed[1].roller.forward;
G_IO.arDO[iReM*4+1].Ch[2]	:= GVL.rem[iReM].infeed[1].roller.backward;
G_IO.arDO[iReM*4+1].Ch[3]	:= GVL.rem[iReM].outfeed[1].roller.Power;
G_IO.arDO[iReM*4+1].Ch[4]	:= GVL.rem[iReM].outfeed[1].roller.forward;
G_IO.arDO[iReM*4+1].Ch[5]	:= GVL.rem[iReM].outfeed[1].roller.backward;
G_IO.arDO[iReM*4+1].Ch[6]	:= GVL.rem[iReM].lift[1].roller.Power;
G_IO.arDO[iReM*4+1].Ch[7]	:= GVL.rem[iReM].lift[1].roller.forward;
G_IO.arDO[iReM*4+1].Ch[8]	:= GVL.rem[iReM].lift[1].roller.backward;
G_IO.arDO[iReM*4+1].Ch[9]	:= GVL.rem[iReM].lift[1].power_axis;
G_IO.arDO[iReM*4+2].Ch[12]	:= GVL.rem[iReM].infeed[1].valve_stopper.extend;
G_IO.arDO[iReM*4+2].Ch[13]	:= GVL.rem[iReM].infeed[1].valve_stopper.retract;
G_IO.arDO[iReM*4+2].Ch[14]	:= GVL.rem[iReM].lift[1].valve_perturbation[0].extend;
G_IO.arDO[iReM*4+3].Ch[0]	:= GVL.rem[iReM].lift[1].valve_perturbation[1].extend;
G_IO.arDO[iReM*4+3].Ch[2]	:= GVL.rem[iReM].lift[1].valve_perturbation[2].extend;
G_IO.arDO[iReM*4+3].Ch[4]	:= GVL.rem[iReM].lift[1].valve_perturbation[3].extend;
G_IO.arDO[iReM*4+3].Ch[6]	:= GVL.rem[iReM].lift[1].valve_clamp.extend;
G_IO.arDO[iReM*4+3].Ch[7]	:= GVL.rem[iReM].lift[1].valve_clamp.retract;

END_FUNCTION_BLOCK

// ---- POUs/FB_remAxisMapping.TcPOU
FUNCTION_BLOCK FB_remAxisMapping
VAR_INPUT
	iReM	: INT;
	iLift	: INT;
	//sNetID	: STRING;
	nSlaveAddr : UINT;
END_VAR
VAR_OUTPUT
END_VAR
VAR
END_VAR

//========== Lift0 Axis Config ==========
GVL.rem[iReM].lift[iLift].mcAxis
(
	ZSN		:= GVL.rem[iReM].lift[iLift].limit_sensor[2] OR GVL.rem[iReM].lift[iLift].st_mcAxis.xHoming,
	ZSP		:= GVL.rem[iReM].lift[iLift].limit_sensor[1]	OR GVL.rem[iReM].lift[iLift].st_mcAxis.xHoming,
	IN_OUT	:= GVL.rem[iReM].lift[iLift].st_mcAxis, 
	AXIS	:= GVL.rem[iReM].lift[iLift].Axisref, 
);
GVL.rem[iReM].lift[iLift].st_mcAxis.bPosSensorShow	:= TRUE;
GVL.rem[iReM].lift[iLift].st_mcAxis.bNegSensorShow	:= TRUE;
GVL.rem[iReM].lift[iLift].st_mcAxis.bStopButtonShow	:= TRUE;
GVL.rem[iReM].lift[iLift].st_mcAxis.rMaxAcceleration	:= 50000;
GVL.rem[iReM].lift[iLift].st_mcAxis.rMaxDeceleration	:= 50000;
GVL.rem[iReM].lift[iLift].st_mcAxis.rMaxJerk			:= 500000;
GVL.rem[iReM].lift[iLift].st_mcAxis.rAcceleration	:= 2500;
GVL.rem[iReM].lift[iLift].st_mcAxis.rDeceleration	:= 2500;
GVL.rem[iReM].lift[iLift].st_mcAxis.rJerk			:= 12500;
GVL.rem[iReM].lift[iLift].st_mcAxis.rMaxVelocity		:= 100;
GVL.rem[iReM].lift[iLift].st_mcAxis.rMaxDistance		:= 50;
GVL.rem[iReM].lift[iLift].st_mcAxis.bPosSen	:= GVL.rem[iReM].lift[iLift].limit_sensor[1] ;
GVL.rem[iReM].lift[iLift].st_mcAxis.bNegSen	:= GVL.rem[iReM].lift[iLift].limit_sensor[2] ;
GVL.rem[iReM].lift[iLift].st_mcAxis.mcHome.bCalibrationCam	:= GVL.rem[iReM].lift[iLift].limit_sensor[0];
GVL.rem[iReM].lift[iLift].st_mcAxis.bPositionSensor	:= GVL.rem[iReM].lift[iLift].limit_sensor[0];
GVL.rem[iReM].lift[iLift].st_mcAxis.bdirFW	:= TRUE;
GVL.rem[iReM].lift[iLift].st_mcAxis.rSetPos	:= 0;
GVL.rem[iReM].lift[iLift].st_mcAxis.sNetID := '192.168.11.159.1.2';
GVL.rem[iReM].lift[iLift].st_mcAxis.nSlaveAddr	:= nSlaveAddr;

END_FUNCTION_BLOCK

// ---- POUs/FB_rmIOmapping.TcPOU
FUNCTION_BLOCK FB_rmIOmapping
VAR_INPUT
	iRm	: INT;
END_VAR
VAR_OUTPUT
END_VAR
	
VAR
	offset	: INT;
	rTrig_power_inConv	: R_TRIG;
	fTrig_power_inConv	: F_TRIG;
	rTrig_power_outConv	: R_TRIG;
	fTrig_power_outConv	: F_TRIG;
	
END_VAR

offset	:= 50+iRm*5;
//pm[odd]
GVL.pm[iRm*2].buffer[0].contractor_axis				:= G_IO.arDI[offset].Ch[0];
GVL.pm[iRm*2].buffer[0].axis_sensor					:= G_IO.arDI[offset].Ch[1];
GVL.pm[iRm*2].buffer[0].surfae_slot_0				:= G_IO.arDI[offset].Ch[2];
GVL.pm[iRm*2].buffer[0].surfae_slot_1				:= G_IO.arDI[offset].Ch[3];
GVL.pm[iRm*2].buffer[0].surfae_slot_2				:= G_IO.arDI[offset].Ch[4];
GVL.pm[iRm*2].buffer[0].above_fixture_light_curtain	:= G_IO.arDI[offset].Ch[5];
GVL.pm[iRm*2].buffer[0].button						:= G_IO.arDI[offset].Ch[6];
GVL.pm[iRm*2].buffer[0].locked						:= G_IO.arDI[offset].Ch[7];
GVL.pm[iRm*2].buffer[0].magnet_locked				:= G_IO.arDI[offset].Ch[8];
GVL.pm[iRm*2].buffer[1].contractor_axis				:= G_IO.arDI[offset].Ch[9];
GVL.pm[iRm*2].buffer[1].axis_sensor					:= G_IO.arDI[offset].Ch[10];
GVL.pm[iRm*2].buffer[1].surfae_slot_0				:= G_IO.arDI[offset].Ch[11];
GVL.pm[iRm*2].buffer[1].surfae_slot_1				:= G_IO.arDI[offset].Ch[12];
GVL.pm[iRm*2].buffer[1].surfae_slot_2				:= G_IO.arDI[offset].Ch[13];
GVL.pm[iRm*2].buffer[1].above_fixture_light_curtain	:= G_IO.arDI[offset].Ch[14];
GVL.pm[iRm*2].buffer[1].button						:= G_IO.arDI[offset].Ch[15];
GVL.pm[iRm*2].buffer[1].locked						:= G_IO.arDI[offset+1].Ch[0];
GVL.pm[iRm*2].buffer[1].magnet_locked				:= G_IO.arDI[offset+1].Ch[1];
GVL.pm[iRm*2].contactor_robot						:= G_IO.arDI[offset+1].Ch[2];
GVL.pm[iRm*2].inConv.valve[0].extended				:= G_IO.arDI[offset+1].Ch[3];
GVL.pm[iRm*2].inConv.valve[0].retracted				:= G_IO.arDI[offset+1].Ch[4];
GVL.pm[iRm*2].inConv.valve[1].extended				:= G_IO.arDI[offset+1].Ch[5];
GVL.pm[iRm*2].inConv.valve[1].retracted				:= G_IO.arDI[offset+1].Ch[6];
GVL.pm[iRm*2].inConv.valve[2].extended				:= G_IO.arDI[offset+1].Ch[7];
GVL.pm[iRm*2].inConv.valve[2].retracted				:= G_IO.arDI[offset+1].Ch[8];
GVL.pm[iRm*2].outConv.photo_sensor[0]				:= G_IO.arDI[offset+1].Ch[9];
GVL.pm[iRm*2].outConv.photo_sensor[1]				:= G_IO.arDI[offset+1].Ch[10];
GVL.pm[iRm*2].outConv.valve[0].extended				:= G_IO.arDI[offset+1].Ch[11];
GVL.pm[iRm*2].outConv.valve[0].retracted			:= G_IO.arDI[offset+1].Ch[12];
GVL.pm[iRm*2].outConv.valve[1].extended				:= G_IO.arDI[offset+1].Ch[13];
GVL.pm[iRm*2].outConv.valve[1].retracted			:= G_IO.arDI[offset+1].Ch[14];

G_IO.arDO[offset].Ch[0]	:= GVL.pm[iRm*2].buffer[0].power_axis;
G_IO.arDO[offset].Ch[1]	:= GVL.pm[iRm*2].buffer[0].magnet;
G_IO.arDO[offset].Ch[2]	:= GVL.pm[iRm*2].buffer[1].power_axis;
G_IO.arDO[offset].Ch[3]	:= GVL.pm[iRm*2].buffer[1].magnet;
G_IO.arDO[offset].Ch[4]	:= GVL.pm[iRm*2].power_robot;
G_IO.arDO[offset].Ch[12]	:= GVL.pm[iRm*2].buffer[0].lamp_button;
G_IO.arDO[offset].Ch[13]	:= GVL.pm[iRm*2].buffer[1].lamp_button;
	
G_IO.arDO[offset+2].Ch[0]	:= GVL.pm[iRm*2].inConv.valve[0].extend;
G_IO.arDO[offset+2].Ch[2]	:= GVL.pm[iRm*2].inConv.valve[1].extend;
G_IO.arDO[offset+2].Ch[4]	:= GVL.pm[iRm*2].inConv.valve[2].extend;
G_IO.arDO[offset+2].Ch[6]	:= GVL.pm[iRm*2].outConv.valve[0].extend;
G_IO.arDO[offset+2].Ch[8]	:= GVL.pm[iRm*2].outConv.valve[1].extend;




//pm[even]
GVL.pm[iRm*2+1].buffer[0].contractor_axis				:= G_IO.arDI[offset+2].Ch[0];
GVL.pm[iRm*2+1].buffer[0].axis_sensor					:= G_IO.arDI[offset+2].Ch[1];
GVL.pm[iRm*2+1].buffer[0].surfae_slot_0				:= G_IO.arDI[offset+2].Ch[2];
GVL.pm[iRm*2+1].buffer[0].surfae_slot_1				:= G_IO.arDI[offset+2].Ch[3];
GVL.pm[iRm*2+1].buffer[0].surfae_slot_2				:= G_IO.arDI[offset+2].Ch[4];
GVL.pm[iRm*2+1].buffer[0].above_fixture_light_curtain	:= G_IO.arDI[offset+2].Ch[5];
GVL.pm[iRm*2+1].buffer[0].button						:= G_IO.arDI[offset+2].Ch[6];
GVL.pm[iRm*2+1].buffer[0].locked						:= G_IO.arDI[offset+2].Ch[7];
GVL.pm[iRm*2+1].buffer[0].magnet_locked				:= G_IO.arDI[offset+2].Ch[8];
GVL.pm[iRm*2+1].buffer[1].contractor_axis				:= G_IO.arDI[offset+2].Ch[9];
GVL.pm[iRm*2+1].buffer[1].axis_sensor					:= G_IO.arDI[offset+2].Ch[10];
GVL.pm[iRm*2+1].buffer[1].surfae_slot_0				:= G_IO.arDI[offset+2].Ch[11];
GVL.pm[iRm*2+1].buffer[1].surfae_slot_1				:= G_IO.arDI[offset+2].Ch[12];
GVL.pm[iRm*2+1].buffer[1].surfae_slot_2				:= G_IO.arDI[offset+2].Ch[13];
GVL.pm[iRm*2+1].buffer[1].above_fixture_light_curtain	:= G_IO.arDI[offset+2].Ch[14];
GVL.pm[iRm*2+1].buffer[1].button						:= G_IO.arDI[offset+2].Ch[15];
GVL.pm[iRm*2+1].buffer[1].locked						:= G_IO.arDI[offset+3].Ch[0];
GVL.pm[iRm*2+1].buffer[1].magnet_locked				:= G_IO.arDI[offset+3].Ch[1];
GVL.pm[iRm*2+1].contactor_robot						:= G_IO.arDI[offset+3].Ch[2];
GVL.pm[iRm*2+1].inConv.valve[0].extended				:= G_IO.arDI[offset+3].Ch[3];
GVL.pm[iRm*2+1].inConv.valve[0].retracted				:= G_IO.arDI[offset+3].Ch[4];
GVL.pm[iRm*2+1].inConv.valve[1].extended				:= G_IO.arDI[offset+3].Ch[5];
GVL.pm[iRm*2+1].inConv.valve[1].retracted				:= G_IO.arDI[offset+3].Ch[6];
GVL.pm[iRm*2+1].inConv.valve[2].extended				:= G_IO.arDI[offset+3].Ch[7];
GVL.pm[iRm*2+1].inConv.valve[2].retracted				:= G_IO.arDI[offset+3].Ch[8];
GVL.pm[iRm*2+1].outConv.photo_sensor[0]				:= G_IO.arDI[offset+3].Ch[9];
GVL.pm[iRm*2+1].outConv.photo_sensor[1]				:= G_IO.arDI[offset+3].Ch[10];
GVL.pm[iRm*2+1].outConv.valve[0].extended				:= G_IO.arDI[offset+3].Ch[11];
GVL.pm[iRm*2+1].outConv.valve[0].retracted			:= G_IO.arDI[offset+3].Ch[12];
GVL.pm[iRm*2+1].outConv.valve[1].extended				:= G_IO.arDI[offset+3].Ch[13];
GVL.pm[iRm*2+1].outConv.valve[1].retracted			:= G_IO.arDI[offset+3].Ch[14];

G_IO.arDO[offset].Ch[5]	:= GVL.pm[iRm*2+1].buffer[0].power_axis;
G_IO.arDO[offset].Ch[6]	:= GVL.pm[iRm*2+1].buffer[0].magnet;
G_IO.arDO[offset].Ch[7]	:= GVL.pm[iRm*2+1].buffer[1].power_axis;
G_IO.arDO[offset].Ch[8]	:= GVL.pm[iRm*2+1].buffer[1].magnet;
G_IO.arDO[offset].Ch[9]	:= GVL.pm[iRm*2+1].power_robot;
G_IO.arDO[offset].Ch[14]	:= GVL.pm[iRm*2+1].buffer[0].lamp_button;
G_IO.arDO[offset].Ch[15]	:= GVL.pm[iRm*2+1].buffer[1].lamp_button;
	
G_IO.arDO[offset+2].Ch[10]	:= GVL.pm[iRm*2+1].inConv.valve[0].extend;
G_IO.arDO[offset+2].Ch[12]	:= GVL.pm[iRm*2+1].inConv.valve[1].extend;
G_IO.arDO[offset+2].Ch[14]	:= GVL.pm[iRm*2+1].inConv.valve[2].extend;
G_IO.arDO[offset+3].Ch[0]	:= GVL.pm[iRm*2+1].outConv.valve[0].extend;
G_IO.arDO[offset+3].Ch[2]	:= GVL.pm[iRm*2+1].outConv.valve[1].extend;	

GVL.pm[iRm*2].contactor_inConv			:= G_IO.arDI[offset+4].Ch[0];//pm[0] and pm[1]
GVL.pm[iRm*2].contactor_outConv			:= G_IO.arDI[offset+4].Ch[1];//pm[0] and pm[1]
GVL.pm[iRm*2+1].contactor_inConv			:= G_IO.arDI[offset+4].Ch[0];//pm[0] and pm[1]
GVL.pm[iRm*2+1].contactor_outConv			:= G_IO.arDI[offset+4].Ch[1];//pm[0] and pm[1]

rTrig_power_inConv(CLK:=GVL.pm[iRm*2].power_inConv OR GVL.pm[iRm*2+1].power_inConv);
fTrig_power_inConv(CLK:=GVL.pm[iRm*2].power_inConv OR GVL.pm[iRm*2+1].power_inConv);
rTrig_power_outConv(CLK:=GVL.pm[iRm*2].power_outConv OR GVL.pm[iRm*2+1].power_outConv);
fTrig_power_outConv(CLK:=GVL.pm[iRm*2].power_outConv OR GVL.pm[iRm*2+1].power_outConv);

IF rTrig_power_inConv.Q THEN
	GVL.pm[iRm*2].power_inConv	:= TRUE;
	GVL.pm[iRm*2+1].power_inConv	:= TRUE;
END_IF
IF fTrig_power_inConv.Q THEN
	GVL.pm[iRm*2].power_inConv	:= FALSE;
	GVL.pm[iRm*2+1].power_inConv	:= FALSE;
END_IF
IF rTrig_power_outConv.Q THEN
	GVL.pm[iRm*2].power_outConv	:= TRUE;
	GVL.pm[iRm*2+1].power_outConv	:= TRUE;
END_IF
IF fTrig_power_outConv.Q THEN
	GVL.pm[iRm*2].power_outConv	:= FALSE;
	GVL.pm[iRm*2+1].power_outConv	:= FALSE;
END_IF
G_IO.arDO[offset].Ch[10]	:= GVL.pm[iRm*2].power_inConv OR GVL.pm[iRm*2+1].power_inConv;//pm[0] and pm[1]
G_IO.arDO[offset].Ch[11]	:= GVL.pm[iRm*2].power_outConv OR GVL.pm[iRm*2+1].power_outConv;//pm[0] and pm[1]

END_FUNCTION_BLOCK

// ---- POUs/FB_pmAxisMapping.TcPOU
FUNCTION_BLOCK FB_pmAxisMapping
VAR_INPUT
	iPM	: INT;
	iBuffer	: INT;
	//sNetID	: STRING;
	nSlaveAddr : UINT;
END_VAR
VAR_OUTPUT
END_VAR
VAR
END_VAR

//========== Lift0 Axis Config ==========
GVL.pm[iPM].buffer[iBuffer].mcAxis
(
	ZSN		:= TRUE,
	ZSP		:= TRUE,
	IN_OUT	:= GVL.rem[iPM].lift[iBuffer].st_mcAxis, 
	AXIS	:= GVL.rem[iPM].lift[iBuffer].Axisref, 
);
GVL.pm[iPM].buffer[iBuffer].st_mcAxis.bPosSensorShow	:= FALSE;
GVL.pm[iPM].buffer[iBuffer].st_mcAxis.bNegSensorShow	:= FALSE;
GVL.pm[iPM].buffer[iBuffer].st_mcAxis.bStopButtonShow	:= TRUE;
GVL.pm[iPM].buffer[iBuffer].st_mcAxis.rMaxAcceleration	:= 50000;
GVL.pm[iPM].buffer[iBuffer].st_mcAxis.rMaxDeceleration	:= 50000;
GVL.pm[iPM].buffer[iBuffer].st_mcAxis.rMaxJerk			:= 500000;
GVL.pm[iPM].buffer[iBuffer].st_mcAxis.rAcceleration	:= 2500;
GVL.pm[iPM].buffer[iBuffer].st_mcAxis.rDeceleration	:= 2500;
GVL.pm[iPM].buffer[iBuffer].st_mcAxis.rJerk			:= 12500;
GVL.pm[iPM].buffer[iBuffer].st_mcAxis.rMaxVelocity		:= 100;
GVL.pm[iPM].buffer[iBuffer].st_mcAxis.rMaxDistance		:= 50;
GVL.pm[iPM].buffer[iBuffer].st_mcAxis.bPosSen	:= TRUE ;
GVL.pm[iPM].buffer[iBuffer].st_mcAxis.bNegSen	:= TRUE ;
GVL.pm[iPM].buffer[iBuffer].st_mcAxis.mcHome.bCalibrationCam	:= GVL.pm[iPM].buffer[iBuffer].axis_sensor;
GVL.pm[iPM].buffer[iBuffer].st_mcAxis.bPositionSensor	:= GVL.pm[iPM].buffer[iBuffer].axis_sensor;
GVL.pm[iPM].buffer[iBuffer].st_mcAxis.bdirFW	:= TRUE;
GVL.pm[iPM].buffer[iBuffer].st_mcAxis.rSetPos	:= 0;
GVL.pm[iPM].buffer[iBuffer].st_mcAxis.sNetID := '192.168.11.159.1.2';
GVL.pm[iPM].buffer[iBuffer].st_mcAxis.nSlaveAddr	:= nSlaveAddr;

END_FUNCTION_BLOCK

// ---- POUs/FB_axisCtrl.TcPOU
FUNCTION_BLOCK FB_axisCtrl
VAR_INPUT
	
END_VAR
VAR_OUTPUT
END_VAR
VAR_IN_OUT     
	stAxisCtrl	:ST_axisCtrl; 	
	IN_OUT 		: ST_MotionAxis_MC	;//struct for each axis
END_VAR
VAR

END_VAR

//add timeout for this fuction block
CASE stAxisCtrl.iCmd OF
	0:
		IN_OUT.mcReset.Execute	:= FALSE;
		IN_OUT.mcStop.Execute	:= FALSE	;
	1:
		IN_OUT.mcPower.Enable	:= TRUE;
		stAxisCtrl.iCmd	:= 0;
	2:
		IN_OUT.mcPower.Enable	:= FALSE;
		stAxisCtrl.iCmd	:= 0;	
	3:
		IN_OUT.mcReset.Execute	:= TRUE;
		stAxisCtrl.iCmd	:= 0;
	4:
		IN_OUT.mcStop.Execute	:= TRUE;
		stAxisCtrl.iCmd	:= 0;	
	5: 
		IN_OUT.mcMoveAbsolute.Execute := TRUE;
		IN_OUT.rActualPosSet	:= stAxisCtrl.rPosition;
		IN_OUT.rVelocitySet	:= stAxisCtrl.iSpeed;
		IF IN_OUT.mcMoveAbsolute.Done THEN
			stAxisCtrl.iCmd	:= 0;
		END_IF
END_CASE;
stAxisCtrl.iStatus := stAxisCtrl.iCmd;

END_FUNCTION_BLOCK

// ---- GVLs/kitting deca/axis/FB_MotionAxis_MC.TcPOU
FUNCTION_BLOCK FB_MotionAxis_MC

VAR_INPUT
	ZSN	   			: BOOL												;
	ZSP				: BOOL												; 
	Exceeding_us			: INT;
	sNameAxis				: STRING [40];

END_VAR         	
                	
VAR  
	rtFirstCycle	: R_TRIG;						
	mcHomeAxis		: 	MC_HomeAxis						;//ADD BY EVAN 
	sAxisName		: STRING											;//Axis name          	
	xPlus			: BOOL												;	
	xMinus			: BOOL												;
	bDone			: BOOL												;	

// Variables for Hard Stop Homing	                        			
	iStatehsHomig	: E_HomingSteps := E_HomingSteps.IDLE				;
	rtHome			: R_TRIG											;
	rtHomeReset		: R_TRIG											;
	tonTimeOut		: TON												;
	xTimerStart		: BOOL												;
	bLSDefaultVal	: BOOL												; // Save Def value from driver
	xHomeError		: BOOL												;
// Variables for Force Control          					

	rtForceC		: R_TRIG											;
	rtForceCReset	: R_TRIG											;
	DelMaxPos		: LREAL 											;
	rCurrLimit		: LREAL												;
	StartPos		: LREAL												;
	xForceCError	: BOOL												;
//	Variables for Backlash Compensation
	rLastMove		: LREAL := 1										;
	tonBackComp		: TON												;
	rBacklashPer	: LREAL												;	
	
// Variables for errors
	rtError					:	R_TRIG;
	pTextType				:	POINTER TO STRING;
	sAxisErrorID			:	STRING(10);	
	ErrorMSG				:	STRING[255];

//	Exceeding time measuring
	sysTime					:	GETCPUCOUNTER;//GETSYSTEMTIME;					//	Used to measure execution time.
	uStartTime				:	UDINT;
	uFinishTime				:	UDINT;
	ftimeDiff				:	REAL;
	ton_dly	: TON;
END_VAR         	
                	
VAR_IN_OUT      	
	IN_OUT 			: ST_MotionAxis_MC	;//struct for each axis
	AXIS 			: AXIS_REF			;//Axis obj	
END_VAR

VAR_OUTPUT
	xError			: BOOL				;
	xBusy			: BOOL				;
END_VAR
VAR CONSTANT
	parallelGroupTLName		:	STRING := 'Port_851.TL_Axis_Error';
END_VAR

(* Power options ********************************************************************************************)			
IN_OUT.mcPower(
	Axis				:= AXIS, 
	Enable				:= , 
	Enable_Positive		:= ZSP, 
	Enable_Negative		:= ZSN OR IN_OUT.mcHome.Busy, 
	Override			:= , 
	BufferMode			:= , 
	Options				:= , 
	Status				=> , 
	Busy				=> , 
	Active				=> , 
	Error				=> , 
	ErrorID				=> );
	
(* Halt Mode ********************************************************************************************)	
IN_OUT.mcHalt(
	Axis				:= AXIS, 
	Execute				:= , 
	Deceleration		:= IN_OUT.rDeceleration, 
	Jerk				:= , 
	BufferMode			:= , 
	Options				:= , 
	Done				=> , 
	Busy				=> , 
	Active				=> , 
	CommandAborted		=> , 
	Error				=> , 
	ErrorID				=> );
	
(* Homing ***********************************************************************************************)
IN_OUT.mcHome(
	Axis				:= AXIS, 
	Execute				:= , 
	Position			:= in_out.rFirstpos, 
	HomingMode			:= MC_Direct, 
	BufferMode			:= , 
	Options				:= , 
	bCalibrationCam		:= ,//NOT  ZSN, 
	Done				=> , 
	Busy				=> , 
	Active				=> , 
	CommandAborted		=> , 
	Error				=> , 
	ErrorID				=> );
	
(* JOG **************************************************************************************************)
IN_OUT.mcJog(
	Axis				:= AXIS, 
	JogForward			:= , 
	JogBackwards		:= , 
	Mode				:= E_JogMode.MC_JOGMODE_CONTINOUS, 
	Position			:= , 
	Velocity			:= IN_OUT.rVelocity, 
	Acceleration		:= IN_OUT.rAcceleration, 
	Deceleration		:= IN_OUT.rDeceleration, 
	Jerk				:= IN_OUT.rJerk, 
	Done				=> , 
	Busy				=> , 
	Active				=> , 
	CommandAborted		=> , 
	Error				=> , 
	ErrorID				=> );
	
(* Move Absolute ****************************************************************************************)	
IN_OUT.mcMoveAbsolute(
	Axis				:= AXIS, 
	Execute				:= , 
	Position			:= IN_OUT.rActualPosSet, 
	Velocity			:= IN_OUT.rVelocitySet,     
	Acceleration		:= IN_OUT.rAcceleration, 
	Deceleration		:= IN_OUT.rDeceleration, 
	Jerk				:= IN_OUT.rJerk,         
	BufferMode			:= , 
	Options				:= , 
	Done				=> , 
	Busy				=> , 
	Active				=> , 
	CommandAborted		=> , 
	Error				=> , 
	ErrorID				=> );

	IF IN_OUT.bMoveAbsHMI THEN
		IN_OUT.mcMoveAbsolute.Execute	:= TRUE;
		IN_OUT.rActualPosSet	:= IN_OUT.rActualPosHMI;
		IN_OUT.rVelocitySet		:= IN_OUT.rVeloPers;
	END_IF
(* Move Relative *********************************************************************************************************)
IN_OUT.mcMoveRelative(
	Axis				:= AXIS, 
	Execute				:= , 
	Distance			:= IN_OUT.rPosition + IN_OUT.rBacklashvalue, 
	Velocity			:= IN_OUT.rVelocity,      
	Acceleration		:= IN_OUT.rAcceleration,  
	Deceleration		:= IN_OUT.rDeceleration,  
	Jerk				:= IN_OUT.rJerk,          
	BufferMode			:= ,
	Options				:= , 
	Done				=> bDone, 
	Busy				=> , 
	Active				=> , 
	CommandAborted		=> , 
	Error				=> , 
	ErrorID				=> );
	
(* Move Velocity *********************************************************************************************************)
	
IN_OUT.mcMoveVelocity(
	Axis				:=	AXIS,
	Execute				:=	,
	Velocity			:=	IN_OUT.rVelocity,
	Acceleration		:=	IN_OUT.rAcceleration,
	Deceleration		:=	IN_OUT.rDeceleration,
	Jerk				:=	IN_OUT.rJerk,
	Direction			:=	IN_OUT.axisDirection,
	BufferMode			:=	,
	Options				:=	,
	InVelocity			=>	,
	Busy				=>	,
	Active				=>	,
	CommandAborted		=>	,
	Error				=>	,
	ErrorID				=>	);
	
(**)	
IN_OUT.mcReadStatus(
	Axis				:= AXIS, 
	Enable				:= TRUE, 
	Valid				=> , 
	Busy				=> , 
	Error				=> , 
	ErrorID				=> , 
	ErrorStop			=> , 
	Disabled			=> , 
	Stopping			=> , 
	StandStill			=> , 
	DiscreteMotion		=> , 
	ContinuousMotion	=> , 
	SynchronizedMotion	=> , 
	Homing				=> , 
	ConstantVelocity	=> , 
	Accelerating		=> , 
	Decelerating		=> , 
	Status				=> );
	
(* Reset ************************************************************************************************)
IN_OUT.mcReset(
	Axis				:= AXIS, 
	Execute				:= , 
	Done				=> , 
	Busy				=> , 
	Error				=> , 
	ErrorID				=> );
	
(* Stop *************************************************************************************************)
IN_OUT.mcStop(
	Axis				:= AXIS, 
	Execute				:= , 
	Deceleration		:= , 
	Jerk				:= , 
	Options				:= , 
	Done				=> , 
	Busy				=> , 
	Active				=> , 
	CommandAborted		=> , 
	Error				=> , 
	ErrorID				=> );

(* Set Position *************************************************************************************************)
in_out.mcSetpoint(
	Axis			 := AXIS, 
	Execute			 := , 
	Position		 := IN_OUT.rSetPos, 
	Mode			 := , 
	Options			 := , 
	Done			 => , 
	Busy			 => , 
	Error			 => , 
	ErrorID			 => );


(* write status *************************************************************************************************)
IN_OUT.mcWriteBoolParameter(
	Axis			:= 	AXIS, 
	Execute:= 				, 
	ParameterNumber:= 		, 
	Value:= , 
	Done=> , 
	Busy=> , 
	Error=> , 
	ErrorID=> );

(* Read status *************************************************************************************************)
IN_OUT.mcReadBoolParameter(
	Axis:= AXIS, 
	Enable:= , 
	ParameterNumber:= , 
	ReadMode:= , 
	Valid=> , 
	Busy=> , 
	Error=> , 
	ErrorID=> , 
	Value=> );	

(*Read Actualposition***************************************************************)
IN_OUT.mcReadActualPosition(
	Axis:= AXIS, 
	Enable:= TRUE, 
	Valid=> , 
	Busy=> , 
	Error=> , 
	ErrorID=> , 
	Position=> IN_OUT.rActualPos );   
(*COE write**************************************************************************)	

IN_OUT.CoeWrt(
	sNetId:= IN_OUT.sNetID, 
	nSlaveAddr:= IN_OUT.nSlaveAddr, 
	nSubIndex:= IN_OUT.nSubIndex, 
	nIndex:= IN_OUT.nIndex, 
	pSrcBuf:= ADR(IN_OUT.iSdoWrite), 
	cbBufLen:= SIZEOF(IN_OUT.iSdoWrite), 
	bExecute:= , 
	tTimeout:= , 
	bBusy=> , 
	bError=> , 
	nErrId=> );
	ton_dly(PT:=T#100MS);
CASE IN_OUT.iCoeWrt OF 
	0:
		IN_OUT.CoeWrt.bExecute := FALSE;
	1:
		IN_OUT.CoeWrt.bExecute := TRUE;
		IN_OUT.nIndex	:= 16#2005;
		IN_OUT.nSubIndex	:= 16#1F;
		IN_OUT.iSdoWrite	:= 6;//clear encoder and set current position as origin
		IN_OUT.iCoeWrt	:= 10;
	2:
		IN_OUT.CoeWrt.bExecute := TRUE;
		IN_OUT.nIndex	:= 16#2002;
		IN_OUT.nSubIndex	:= 16#02;
		IN_OUT.iSdoWrite	:= 1;//linear mode
		IN_OUT.iCoeWrt	:= 10;
	3:
		IN_OUT.CoeWrt.bExecute := TRUE;
		IN_OUT.nIndex	:= 16#2002;
		IN_OUT.nSubIndex	:= 16#02;
		IN_OUT.iSdoWrite	:= 2;//rotate mode
		IN_OUT.iCoeWrt	:= 10;
	4:
		IN_OUT.CoeWrt.bExecute := TRUE;
		IN_OUT.nIndex	:= 16#2004;
		IN_OUT.nSubIndex	:= 16#06;
		IN_OUT.iSdoWrite	:= 1;//breaker on
		IN_OUT.iCoeWrt	:= 10;
	5:
		IN_OUT.CoeWrt.bExecute := TRUE;
		IN_OUT.nIndex	:= 16#2004;
		IN_OUT.nSubIndex	:= 16#06;
		IN_OUT.iSdoWrite	:= 0;//breaker off
		IN_OUT.iCoeWrt	:= 10;		
	10:		
		IN_OUT.iCoeWrt	:= 0;
END_CASE







	(*mcHomeAxis***************************************************************)
	mcHomeAxis(
		xExecute:= , 
		xReset:= , 
		InOut:=IN_OUT , 
		xRedy=> , 
		xBusy=> , 
		xDone=> , 
		xError=> ); 
	                                                                                                              	
(******************************************************************************************************************)
	
(**error flag**)
	xError := IN_OUT.mcReadStatus.Error OR xHomeError OR IN_OUT.mcMoveAbsolute.Error ;	
	rtError(CLK:= (IN_OUT.mcReadStatus.ErrorID <> 0) AND NOT IN_OUT.xMuteAxisErrorMessages);
	
(*************************** READ ERROR FROM DRIVE *************************)
rtFirstCycle(CLK:= TRUE);
sysTime(cpuCntLoDW => uStartTime);	
sysTime(cpuCntLoDW => uFinishTime);
//M_CheckExceedingTime();

(*************************** GET AXIS ERROR MESSAGE *************************)	
	
	IF rtError.Q THEN
	sAxisErrorID	:=	TO_STRING(IN_OUT.mcReadStatus.ErrorID);
	END_IF
(**remember the Velocity**) 
	IF IN_OUT.rVeloPers <> 0 THEN 
		IN_OUT.rVelocity:= IN_OUT.rVeloPers;
	ELSE 
		IN_OUT.rVeloPers := IN_OUT.rVelocity;	
	END_IF	
(**remember the Acceleration**)
	IF IN_OUT.rAccPers <> 0 THEN 
		IN_OUT.rAcceleration:= IN_OUT.rAccPers;
	ELSE 
		IN_OUT.rAccPers := IN_OUT.rAcceleration;		
	END_IF	
(**remember the Deceleration**)
	IF IN_OUT.rDecPers <> 0 THEN 
		IN_OUT.rDeceleration:= IN_OUT.rDecPers;
	ELSE 
		IN_OUT.rDecPers := IN_OUT.rDeceleration;		
	END_IF
(**False all Executions if function done or error**)
	IF IN_OUT.mcMoveRelative.Done OR IN_OUT.mcMoveRelative.Error OR IN_OUT.mcReset.Busy THEN 
		IN_OUT.mcMoveRelative.Execute := FALSE;
	END_IF

	IF IN_OUT.mcMoveVelocity.Error OR IN_OUT.mcReset.Busy OR IN_OUT.mcMoveVelocity.Busy THEN 
		IN_OUT.mcMoveVelocity.Execute := FALSE;
	END_IF
	
	IF IN_OUT.mcSetpoint.done OR IN_OUT.mcSetpoint.Error THEN
		IN_OUT.mcSetpoint.Execute := FALSE;
	END_IF
	
    IF  IN_OUT.mcMoveAbsolute.Done OR IN_OUT.mcMoveAbsolute.Error OR IN_OUT.mcReset.Busy THEN 
		IN_OUT.mcMoveAbsolute.Execute := FALSE;
	END_IF
 
	 IF IN_OUT.mcHome.Done OR IN_OUT.mcHome.Error THEN 
		IN_OUT.mcHome.Execute := FALSE;
	END_IF
	
	IF IN_OUT.mcStop.Done OR IN_OUT.mcStop.Error THEN 
		IN_OUT.mcStop.Execute := FALSE;
	END_IF
	
	IF IN_OUT.mcReset.Done OR IN_OUT.mcReset.Error THEN 
		IN_OUT.mcReset.Execute := FALSE;
	END_IF
			
	IF IN_OUT.mcReadBoolParameter.Valid OR IN_OUT.mcReadBoolParameter.Error THEN 
		IN_OUT.mcReadBoolParameter.Enable := FALSE;
	END_IF	
	
	IF IN_OUT.mcWriteBoolParameter.Done OR IN_OUT.mcWriteBoolParameter.Error THEN 
		IN_OUT.mcWriteBoolParameter.Execute	:= FALSE;
	END_IF	
		

	
	
	
(**Save done state into temp variable**)	
	
	IF IN_OUT.mcMoveAbsolute.Done THEN
		IN_OUT.xMoveABSDone := TRUE;
	END_IF	
	
	IF IN_OUT.mcMoveRelative.Done THEN
		IN_OUT.xMoveRelDone := TRUE;
	END_IF

PROPERTY P_AxisName : STRING
SET
sAxisName := P_AxisName;
END_SET
END_PROPERTY

PROPERTY P_CurrLimit : LREAL
SET
rCurrLimit := P_CurrLimit;
END_SET
END_PROPERTY

PROPERTY P_DelMaxPos : LREAL
SET
DelMaxPos := P_DelMaxPos;
END_SET
END_PROPERTY

PROPERTY P_ForceCError : BOOL
GET
P_ForceCError := xForceCError;
END_GET
END_PROPERTY

PROPERTY P_hsHomingError : BOOL
GET
P_hsHomingError := xHomeError;
END_GET
END_PROPERTY

PROPERTY P_StartPos : LREAL
SET
StartPos := P_StartPos;
END_SET
END_PROPERTY

END_FUNCTION_BLOCK

// ---- GVLs/kitting deca/axis/MC_HomeAxis.TcPOU
FUNCTION_BLOCK MC_HomeAxis
VAR_INPUT
	xExecute		: BOOL;
	xReset			: BOOL;
END_VAR

VAR
	eStates 		: E_HomingSteps :=E_HomingSteps.IDLE;
	rtHomeStart		: R_TRIG;
	rtHomeReset		: R_TRIG;
	ton_delay		: TON;
	bError			: BOOL;	
END_VAR
VAR_IN_OUT
	InOut		: ST_MotionAxis_MC;
END_VAR
VAR_OUTPUT
	xRedy		: BOOL;
	xBusy		: BOOL;
	xDone		: BOOL;
	xError		: BOOL;
END_VAR

rtHomeStart(CLK:=xExecute);
rtHomeReset(CLK:=xReset);
ton_delay(PT:= T#2S);

IF rtHomeStart.Q THEN
	eStates := E_HomingSteps.START;
END_IF
IF rtHomeReset.Q THEN
	eStates := E_HomingSteps.IDLE;
END_IF
IF InOut.mcStop.Execute THEN
	eStates := E_HomingSteps.ERROR;
END_IF
CASE eStates OF
		E_HomingSteps.IDLE:// WAIT FOR REQUEST	
	//Wait for Reset
		IF rtHomeReset.Q THEN
			InOut.mcReset.Execute := TRUE;
			InOut.mcJog.JogForward :=FALSE;
			InOut.mcJog.JogBackwards :=FALSE;
			xExecute := FALSE;
			bError := FALSE;
		END_IF	
		InOut.xHoming	:= FALSE;
	E_HomingSteps.INIT:		
		;

	E_HomingSteps.START:
			ton_delay.IN	:= FALSE;
			InOut.xHoming	:= TRUE;
			InOut.rVeloPers :=30;
			IF InOut.bdirFW THEN//first direction
				eStates := E_HomingSteps.JOG_FW;	
			ELSE
				eStates := E_HomingSteps.JOG_BW;	
			END_IF
///////////////////////////////////////////////////////////////////////////	
	E_HomingSteps.JOG_FW:
		IF InOut.bPosSen THEN
			InOut.mcJog.JogForward :=TRUE;			
		ELSE
			InOut.mcJog.JogForward :=FALSE;
			eStates := E_HomingSteps.JOG_BW_DOG;			
		END_IF
	E_HomingSteps.JOG_BW_DOG:
		IF InOut.bPositionSensor THEN
			InOut.mcJog.JogBackwards :=FALSE;
			eStates := E_HomingSteps.FW_DOG_OFF;			
		ELSE
			InOut.mcJog.JogBackwards :=TRUE;
		END_IF	
	E_HomingSteps.FW_DOG_OFF:	
		IF InOut.bPositionSensor THEN
			InOut.mcJog.JogForward := TRUE;
			InOut.rVeloPers	:=	5;						
		ELSE
			InOut.mcJog.JogForward := FALSE;
			eStates := E_HomingSteps.BW_DOG_ON;
		END_IF		
	E_HomingSteps.BW_DOG_ON:
		IF InOut.bPositionSensor THEN
			InOut.mcJog.JogBackwards := FALSE;
			eStates := E_HomingSteps.WAIT;					
		ELSE
			InOut.rVeloPers	:=	2;		
			InOut.mcJog.JogBackwards := TRUE;		
		END_IF		
///////////////////////////////////////////////////////////////////////////	
	E_HomingSteps.JOG_BW:
		IF InOut.bNegSen THEN
			InOut.mcJog.JogBackwards :=TRUE;			
		ELSE
			InOut.mcJog.JogBackwards :=FALSE;
			eStates := E_HomingSteps.JOG_FW_DOG;	
		END_IF
	E_HomingSteps.JOG_FW_DOG:
		IF InOut.bPositionSensor THEN
			InOut.mcJog.JogForward :=FALSE;
			eStates := E_HomingSteps.BW_DOG_OFF;				
		ELSE
			InOut.mcJog.JogForward :=TRUE;
		END_IF	
	E_HomingSteps.BW_DOG_OFF:	
		IF InOut.bPositionSensor THEN
			InOut.mcJog.JogBackwards := TRUE;
			InOut.rVeloPers	:=	5;						
		ELSE
			InOut.mcJog.JogBackwards := FALSE;
			eStates := E_HomingSteps.FW_DOG_ON;
		END_IF		
	E_HomingSteps.FW_DOG_ON:
		IF InOut.bPositionSensor THEN
			InOut.mcJog.JogForward := FALSE;
			eStates := E_HomingSteps.WAIT;					
		ELSE
			InOut.rVeloPers	:=	2;		
			InOut.mcJog.JogForward := TRUE;		
		END_IF		
///////////////////////////////////////////////////////////////////////////
	E_HomingSteps.WAIT:
		ton_delay.IN	:= TRUE;
		IF ton_delay.Q THEN
			eStates := E_HomingSteps.MCHOME;	
		END_IF
	E_HomingSteps.MCHOME:
		IF InOut.mcReadStatus.StandStill THEN
			InOut.mcHome.Execute := TRUE;	
		END_IF
		IF NOT InOut.mcHome.Busy AND InOut.mcHome.Done THEN
			InOut.mcHome.Execute := FALSE;
			eStates := E_HomingSteps.DONE;	
		END_IF		
	E_HomingSteps.DONE:	
		InOut.xHoming	:= FALSE;
		InOut.xHomingDone	:= TRUE;
		InOut.rVeloPers	:=	10;	
		eStates := E_HomingSteps.IDLE;	
		
	E_HomingSteps.ERROR:	
		InOut.mcJog.JogForward :=FALSE;
		InOut.mcJog.JogBackwards :=FALSE;
		IF InOut.mcReadStatus.Error THEN
			InOut.xHomingDone	:= FALSE;
		END_IF		
		eStates := E_HomingSteps.IDLE;	
		
END_CASE

xRedy		:= (eStates = E_HomingSteps.IDLE);
xBusy		:= (eStates > E_HomingSteps.IDLE AND eStates < E_HomingSteps.DONE);
xDone		:= (eStates = E_HomingSteps.DONE );
xError		:= (eStates = E_HomingSteps.ERROR);

END_FUNCTION_BLOCK

// ---- GVLs/kitting deca/FB_DigitalInput.TcPOU
FUNCTION_BLOCK FB_DigitalInput
// Debounce a digital inpit.
VAR_INPUT
	D: BOOL := FALSE;				// Raw sensor input.
	on_ms : DINT := 0;				// Time (ms) signal is true before 'on' is true.
	off_ms : DINT := 0;				// Time (ms) signal is false before 'on' is false.
END_VAR
VAR_OUTPUT
	Q : BOOL := FALSE;	// Debounced signal state.
END_VAR
VAR
	on_timer : TON;
	off_timer : TON;
END_VAR

on_timer.PT := DINT_TO_TIME(on_ms);
off_timer.PT := DINT_TO_TIME(off_ms);

on_timer(IN := D);
off_timer(IN := NOT D);

Q := (on_timer.Q OR Q) AND NOT off_timer.Q;

END_FUNCTION_BLOCK

// ---- GVLs/kitting deca/FB_do.TcPOU
FUNCTION_BLOCK FB_do
VAR_INPUT
END_VAR
VAR_OUTPUT
END_VAR
VAR
END_VAR

END_FUNCTION_BLOCK

// ---- GVLs/kitting deca/FB_PhotoSensor.TcPOU
FUNCTION_BLOCK FB_PhotoSensor
VAR_INPUT
END_VAR
VAR_OUTPUT
END_VAR
VAR
    status: DigitalInputStatus;
	debounced_input: FB_DigitalInput;
END_VAR

METHOD PUBLIC set_status : BOOL
VAR_INPUT
	new_raw_value: BOOL;
	on_ms : DINT := 0;				// Time (ms) signal is true before 'on' is true.
	off_ms : DINT := 50;				// Time (ms) signal is true before 'on' is true.
END_VAR
VAR
	new_debounced_value: BOOL;
END_VAR
debounced_input(D := new_raw_value, on_ms := on_ms, off_ms:= off_ms, Q => new_debounced_value);

IF new_debounced_value = TRUE THEN
	status := DigitalInputStatus.HIGH;
ELSE
	status := DigitalInputStatus.LOW;
END_IF
END_METHOD

END_FUNCTION_BLOCK

// ---- GlobalTextList.TcGTLO
TEXTLIST GlobalTextList
  282 = ''
  206 = '%.2f mm'
  740 = '%.3f mm'
  386 = '%d'
  201 = '%s'
  646 = '%t'
  209 = '+'
  210 = '-'
  153 = '1'
  531 = '11111111111'
  613 = '2'
  265 = '222222'
  171 = '560-2710N/P'
  381 = 'aboveFixture_light_curtain'
  602 = 'Acc'
  843 = 'Actual Position'
  667 = 'axis'
  203 = 'Axis Error '
  89 = 'Belt'
  1107 = 'belt'
  633 = 'belt test'
  117 = 'Belt test'
  411 = 'Belt Test'
  476 = 'belt[0]'
  143 = 'belt[1]'
  1145 = 'belt[2]'
  388 = 'Breaker'
  808 = 'Breaker OFF'
  486 = 'Breaker ON'
  994 = 'buffer0'
  1091 = 'Buffer0'
  1220 = 'buffer1'
  506 = 'Buffer1'
  183 = 'Buffer[0]'
  1331 = 'Buffer[1]'
  360 = 'buffer_surface_LC_slot_0'
  733 = 'button'
  235 = 'button lamp'
  856 = 'Clear'
  393 = 'cmd'
  981 = 'count'
  349 = 'Dec'
  216 = 'deg/s'
  217 = 'deg/s²'
  662 = 'DOG'
  396 = 'elapse time'
  673 = 'error'
  924 = 'Extend'
  614 = 'extended'
  625 = 'FR test'
  174 = 'FR Test'
  1075 = 'freq'
  841 = 'HOME'
  248 = 'HomeDone'
  986 = 'Infeed[0]'
  112 = 'Infeed[1]'
  886 = 'infeed[].photo_sensor[0]'
  1022 = 'inner_conveyor'
  99 = 'Jerk'
  839 = 'JOG BW'
  840 = 'JOG FW'
  79 = 'LCS0307-E15'
  250 = 'Lift0'
  698 = 'Lift1'
  382 = 'Lift[0]'
  688 = 'Lift[1]'
  1012 = 'locked'
  373 = 'magnet'
  896 = 'magnet locked'
  447 = 'MAIN.iCnt1'
  456 = 'MAIN.tCnt1'
  492 = 'measuring light curtain'
  215 = 'mm/s'
  214 = 'mm/s²'
  207 = 'MOVE ABS'
  569 = 'Move relative'
  524 = 'ms'
  169 = 'NC_contactor'
  205 = 'Neg LS'
  749 = 'Other'
  869 = 'Others'
  530 = 'outer_conveyor'
  162 = 'Outfeed[0]'
  990 = 'Outfeed[1]'
  494 = 'outter_conveyor'
  223 = 'page1'
  737 = 'page2'
  1439 = 'photo_sensor'
  70 = 'photo_sensor[0]'
  865 = 'photo_sensor[1]'
  876 = 'PM'
  413 = 'PM0'
  1418 = 'PM1'
  809 = 'PM2'
  1129 = 'PM3'
  1328 = 'PM4'
  55 = 'PM5'
  859 = 'PM6'
  1156 = 'PM7'
  1732 = 'PM8'
  989 = 'PM9'
  1105 = 'PM_0'
  617 = 'PM_1'
  911 = 'PM_IO'
  204 = 'Pos LS'
  218 = 'power'
  844 = 'Power \nOn'
  359 = 'Power On'
  1449 = 'Power ON'
  755 = 'ReM'
  457 = 'ReM0'
  355 = 'rem0IO_0'
  452 = 'rem0IO_1'
  315 = 'rem0_IO_0'
  86 = 'rem0_IO_1'
  852 = 'ReM1'
  296 = 'ReM2'
  1185 = 'ReM3'
  904 = 'ReM4'
  274 = 'ReM5'
  882 = 'ReM6'
  996 = 'ReM7'
  763 = 'ReM8'
  1106 = 'ReM9'
  1355 = 'ReMIO_0'
  1011 = 'ReMIO_1'
  672 = 'rem_0'
  155 = 'ReM_0'
  88 = 'rem_1'
  795 = 'ReM_1'
  462 = 'Replenishment'
  199 = 'Reset'
  481 = 'Retract'
  934 = 'retracted'
  1226 = 'RFID[0]'
  453 = 'RFID[1]'
  186 = 'robot'
  72 = 'roller'
  983 = 'Set absolute\nencoder as line'
  622 = 'Set absolute\nencoder as linear'
  454 = 'Set absolute\nencoder as rotation'
  606 = 'Set absolute \nencoder as line'
  230 = 'Set absolute encoder\n'
  976 = 'Set absoluteencoder \nas line'
  545 = 'Set Incremental encoder'
  883 = 'Set incremental encoder'
  871 = 'Set incremental encoder \nas line'
  719 = 'Set incremental encoder as line'
  208 = 'Set Point'
  14 = 'Set Pos to 0'
  284 = 'sick measure'
  765 = 'SLC'
  971 = 'slot_0'
  156 = 'slot_1'
  122 = 'slot_2'
  198 = 'Stop'
  336 = 'surface_light_curtain'
  379 = 'time'
  637 = 'valve_clamp'
  1384 = 'valve_inner[0]'
  67 = 'valve_inner[1]'
  1359 = 'valve_inner[2]'
  1180 = 'valve_outer[0]'
  1288 = 'valve_outer[1]'
  728 = 'valve_outter[0]'
  516 = 'valve_perturbation[0]'
  836 = 'valve_perturbation[1]'
  970 = 'valve_perturbation[2]'
  148 = 'valve_perturbation[3]'
  227 = 'valve_stopper'
  200 = 'Velocity'
  403 = 'X'
  404 = 'Y'
  405 = 'Z'
  607 = '计数'
  641 = '计算'
  664 = '页面1'
END_TEXTLIST

// ---- GVLs/kitting deca/axis/AxisHMI_Ex.TcVIS
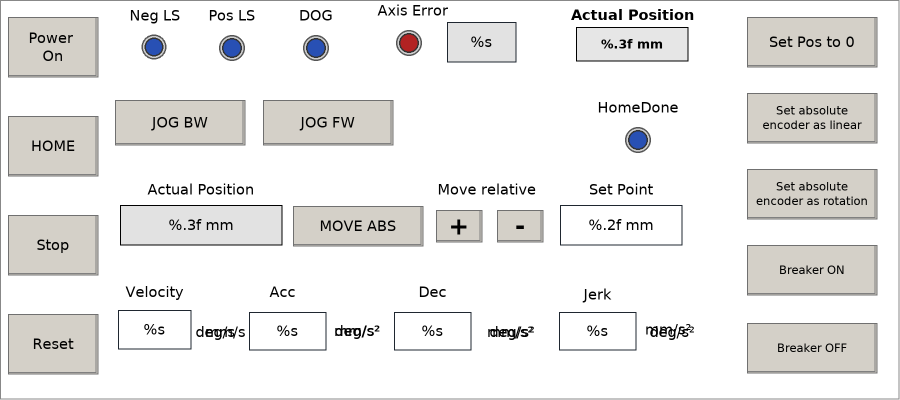
VISUALIZATION AxisHMI_Ex  // 900x400
VAR_IN_OUT
	stAxisHMI	: ST_MotionAxis_MC	;
	mcAxis		: FB_MotionAxis_MC;
	//sAxisName	: STRING			;// Axis Name
	//iAxisID		: INT			;// Axis Id
	xError		: BOOL				;// Axis error flag
END_VAR
    Button (115,100 130x45), "JOG BW", colour toggle: stAxisHMI.mcJog.JogBackwards
        OnMouseDown: execute { stAxisHMI.mcJog.JogBackwards := TRUE; }
        OnMouseUp: execute { stAxisHMI.mcJog.JogBackwards := FALSE; }
    Button (263,100 130x45), "JOG FW", colour toggle: stAxisHMI.mcJog.JogForward
        OnMouseDown: execute { stAxisHMI.mcJog.JogForward := TRUE; }
        OnMouseUp: execute { stAxisHMI.mcJog.JogForward := FALSE; }
    Rectangle (120,205 162x40), "%.3f mm", text variable: stAxisHMI.rActualPosHMI
        OnMouseClick: write the text variable via Default
    Label (141,177 120x25), "Actual Position"
    Button (8,17 90x60), "Power On", colour toggle: stAxisHMI.mcPower.Enable, pressed state: stAxisHMI.mcPower.Enable
        OnMouseClick: toggle stAxisHMI.mcPower.Enable
    Button (8,215 90x60), "Stop", colour toggle: stAxisHMI.mcStop.Execute, invisible if: NOT stAxisHMI.bStopButtonShow
        OnMouseDown: execute { stAxisHMI.mcStop.Execute := TRUE; }
        OnMouseUp: execute { stAxisHMI.mcStop.Execute := FALSE; }
    Button (8,314 90x60), "Reset", colour toggle: stAxisHMI.mcReset.Execute
        OnMouseDown: execute { stAxisHMI.mcReset.Execute := TRUE; }
        OnMouseUp: execute { stAxisHMI.mcReset.Execute := FALSE; }
    Label (111,277 87x30), "Velocity"
    Rectangle (118,310 73x39), "%s", text variable: stAxisHMI.rVeloPers
        OnMouseClick: write the text variable via Default, min 1, max stAxisHMI.rMaxVelocity
    Label (230,277 105x30), "Acc"
    Rectangle (249,312 77x38), "%s", text variable: stAxisHMI.rAcceleration
        OnMouseClick: write stAxisHMI.rAccPers via Default, min 1, max stAxisHMI.rMaxAcceleration
    Lamp1 (139,33 30x28), variable: stAxisHMI.bNegSen, invisible if: NOT stAxisHMI.bNegSensorShow, style: Lamp-Lamp1-Blue
    Label (364,-2 102x25), "Axis Error"
    Rectangle (447,22 69x40), "%s", text variable: stAxisHMI.mcReadStatus.ErrorID
    Lamp1 (394,28 30x30), variable: xError, style: Lamp-Lamp1-Red
    Lamp1 (217,33 30x30), variable: stAxisHMI.bPosSen, invisible if: NOT stAxisHMI.bPosSensorShow, style: Lamp-Lamp1-Blue
    Label (188,3 88x25), "Pos LS", invisible if: NOT stAxisHMI.bPosSensorShow
    Label (111,3 88x25), "Neg LS", invisible if: NOT stAxisHMI.bNegSensorShow
    Rectangle (560,205 122x40), "%.2f mm", text variable: stAxisHMI.rDistance
        OnMouseClick: write the text variable via Default, min 0, max stAxisHMI.rMaxDistance
    Button (293,206 130x40), "MOVE ABS", colour toggle: stAxisHMI.mcMoveAbsolute.Busy, pressed state: stAxisHMI.mcMoveAbsolute.Busy
        OnMouseDown: execute { stAxisHMI.bMoveAbsHMI := TRUE; }
        OnMouseUp: execute { stAxisHMI.bMoveAbsHMI := FALSE; }
    Label (561,177 120x25), "Set Point"
    Button (436,210 46x32), "+", colour toggle: stAxisHMI.mcMoveRelative.Busy, pressed state: stAxisHMI.mcMoveRelative.Busy
        OnMouseDown: execute { stAxisHMI.rPosition := stAxisHMI.rDistance; stAxisHMI.mcMoveRelative.Execute := TRUE; }
        OnMouseUp: execute { stAxisHMI.mcMoveRelative.Execute := FALSE; }
    Button (497,210 46x32), "-", colour toggle: stAxisHMI.mcMoveRelative.Busy, pressed state: stAxisHMI.mcMoveRelative.Busy
        OnMouseDown: execute { stAxisHMI.rPosition := -(stAxisHMI.rDistance); stAxisHMI.mcMoveRelative.Execute := TRUE; }
        OnMouseUp: execute { stAxisHMI.mcMoveRelative.Execute := FALSE; }
    Label (427,177 120x25), "Move relative"
    Label (330,316 55x30), "mm/s²"
    Label (196,317 59x30), "mm/s"
    Label (191,317 49x30), "deg/s", invisible if: NOT stAxisHMI.bUnitDegShow
    Label (328,316 59x30), "deg/s²", invisible if: NOT stAxisHMI.bUnitDegShow
    Label (380,277 105x30), "Dec"
    Rectangle (394,312 77x38), "%s", text variable: stAxisHMI.rDeceleration
        OnMouseClick: write stAxisHMI.rDecPers via Default, min 1, max stAxisHMI.rMaxDeceleration
    Label (483,317 55x30), "mm/s²"
    Label (483,317 59x30), "deg/s²", invisible if: NOT stAxisHMI.bUnitDegShow
    Button (8,116 90x60), "HOME", colour toggle: stAxisHMI.mcHome.Busy
        OnMouseDown: execute { mcAxis.mcHomeAxis.xExecute	:= TRUE; }
        OnMouseUp: execute { mcAxis.mcHomeAxis.xExecute	:= FALSE; }
    Rectangle (559,312 77x38), "%s", text variable: stAxisHMI.rJerk, invisible if: NOT stAxisHMI.bJerkShow
        OnMouseClick: write the text variable via Default, min 0, max stAxisHMI.rMaxJerk
    Label (572,282 51x25), "Jerk", invisible if: NOT stAxisHMI.bJerkShow
    Label (643,317 59x30), "deg/s²", invisible if: NOT stAxisHMI.bUnitDegShow
    Label (641,317 55x25), "mm/s²", invisible if: NOT stAxisHMI.bJerkShow
    Label (557,0 152x30), "Actual Position"
    Rectangle (576,27 112x34), "%.3f mm", text variable: stAxisHMI.rActualPos
    Lamp1 (301,33 30x30), variable: stAxisHMI.bPositionSensor, style: Lamp-Lamp1-Blue
    Label (272,3 88x25), "DOG", invisible if: NOT stAxisHMI.bPosSensorShow
    Lamp1 (623,125 30x30), variable: stAxisHMI.xHomingDone, style: Lamp-Lamp1-Blue
    Label (594,95 88x25), "HomeDone", invisible if: NOT stAxisHMI.bPosSensorShow
    Button (747,17 130x50), "Set Pos to 0", colour toggle: stAxisHMI.CoeWrt.bExecute
        OnMouseDown: execute {
            (*stAxisHMI.CoeWrt.bExecute := TRUE;
            stAxisHMI.nIndex	:= 16#2005;
            stAxisHMI.nSubIndex	:= 16#1F;
            stAxisHMI.iSdoWrite	:= 6;//clear encoder and set current position as origin*)
            stAxisHMI.mcPower.Enable	:= FALSE;
        }
        OnMouseUp: execute { stAxisHMI.iCoeWrt	:= 1; }
    Button (747,93 130x50), "Set absolute encoder as linear", colour toggle: stAxisHMI.CoeWrt.bExecute
        OnMouseDown: execute {
            (*stAxisHMI.CoeWrt.bExecute := TRUE;
            stAxisHMI.nIndex	:= 16#2002;
            stAxisHMI.nSubIndex	:= 16#02;
            stAxisHMI.iSdoWrite	:= 1;//linear mode*)
        }
        OnMouseUp: execute { (*stAxisHMI.CoeWrt.bExecute := FALSE;*) stAxisHMI.iCoeWrt	:= 2; }
    Button (747,169 130x50), "Set absolute encoder as rotation", colour toggle: stAxisHMI.CoeWrt.bExecute
        OnMouseDown: execute {
            (*stAxisHMI.CoeWrt.bExecute := TRUE;
            stAxisHMI.nIndex	:= 16#2002;
            stAxisHMI.nSubIndex	:= 16#02;
            stAxisHMI.iSdoWrite	:= 2;//rotate mode*)
        }
        OnMouseUp: execute { (*stAxisHMI.CoeWrt.bExecute := FALSE;*) stAxisHMI.iCoeWrt	:= 3; }
    Button (747,245 130x50), "Breaker ON", colour toggle: stAxisHMI.CoeWrt.bExecute
        OnMouseDown: execute {
            (*stAxisHMI.CoeWrt.bExecute := TRUE;
            stAxisHMI.nIndex	:= 16#2004;
            stAxisHMI.nSubIndex	:= 16#06;
            stAxisHMI.iSdoWrite	:= 1;//rotate mode*)
        }
        OnMouseUp: execute { (*stAxisHMI.CoeWrt.bExecute := FALSE;*) stAxisHMI.iCoeWrt	:= 4; }
    Button (747,323 130x50), "Breaker OFF", colour toggle: stAxisHMI.CoeWrt.bExecute
        OnMouseDown: execute {
            (*stAxisHMI.CoeWrt.bExecute := TRUE;
            stAxisHMI.nIndex	:= 16#2004;
            stAxisHMI.nSubIndex	:= 16#06;
            stAxisHMI.iSdoWrite	:= 0;//*)
        }
        OnMouseUp: execute { (*stAxisHMI.CoeWrt.bExecute := FALSE;*) stAxisHMI.iCoeWrt	:= 5; }
END_VISUALIZATION

// ---- VISUs/OtherList.TcVIS
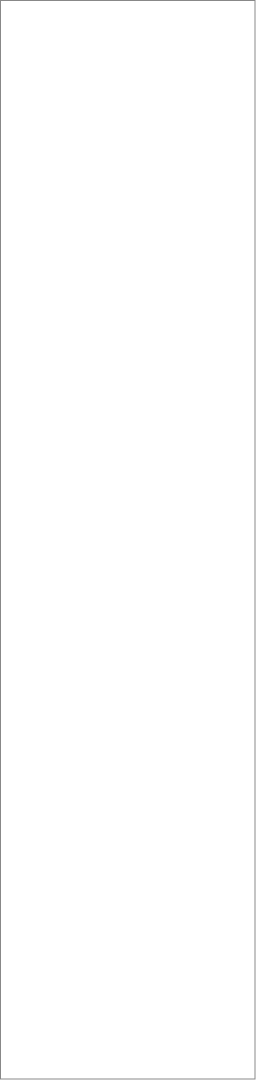
VISUALIZATION OtherList  // 256x1080
    Button (1413,1160 244x110), "ReM0"
        OnMouseDown: execute { G_HMI.iMainFrame  := 0; }
END_VISUALIZATION

// ---- VISUs/visu_PM.TcVIS
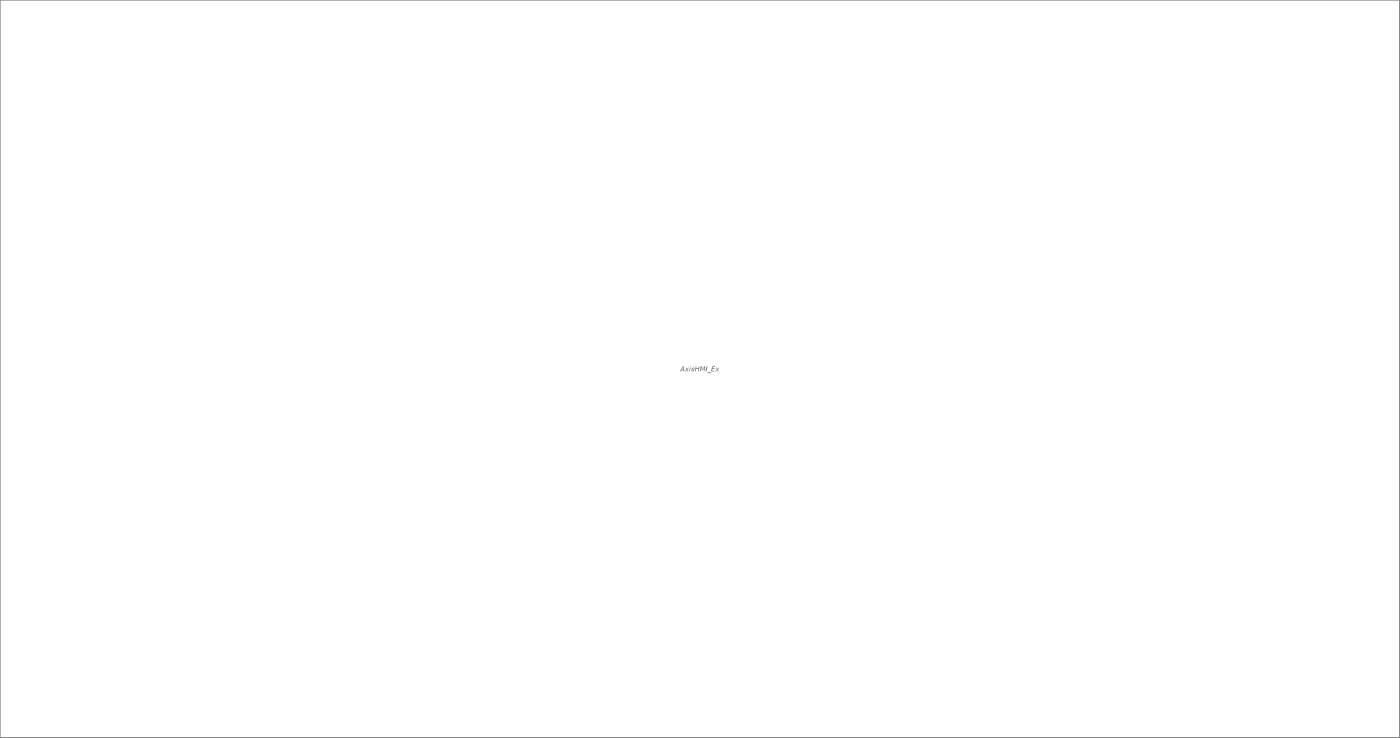
VISUALIZATION visu_PM  // 2048x1080
    TabControl (0,0 2048x1080)
        shows AxisHMI_Ex(stAxisHMI := GVL.pm[G_HMI.iPM].buffer[0].st_mcAxis, mcAxis := GVL.pm[G_HMI.iPM].buffer[0].mcAxis, xError := GVL.pm[G_HMI.iPM].buffer[0].mcAxis.xError)
        shows AxisHMI_Ex(stAxisHMI := GVL.pm[G_HMI.iPM].buffer[1].st_mcAxis, mcAxis := GVL.pm[G_HMI.iPM].buffer[1].mcAxis, xError := GVL.pm[G_HMI.iPM].buffer[1].mcAxis.xError)
        shows v_pm_0(dIO_PM := GVL.pm[G_HMI.iPM])
        shows Axis_HMI(st_axis_HMI := st_mcAxis[EN_Axis.Grip_axis])
        shows v_rem_1(dIO_ReM := GVL.pm[G_HMI.iModule])
        [0]: TabTitle=Buffer0
        [1]: TabTitle=Buffer1
        [6]: TabTitle=Gripper
        [2]: AxisHMI=gantrybase.st_mcAxis[EN_Axis.Z], mcAxis=gantrybase.mcAxis[EN_Axis.Z], Error=gantrybase.mcAxis[EN_Axis.Z].xError
        p699000190: gantrybase.st_mcAxis[EN_Axis.X]
        p2837713833: gantrybase.mcAxis[EN_Axis.Z].sAxisName
        p520277221: gantrybase.mcAxis[EN_Axis.X].xError
        p3331604638: gantrybase.st_mcAxis[EN_Axis.Z]
        p1813558639: gantrybase.mcAxis[EN_Axis.Z].xError
        p1563495665: gantrybase.st_mcAxis[EN_Axis.Y]
        p2070126892: gantrybase.mcAxis[EN_Axis.Y].xError
        p3435970784: gantrybase.mcAxis[EN_Axis.X]
        p2829954345: gantrybase.mcAxis[EN_Axis.Y]
        p3218520426: gantrybase.mcAxis[EN_Axis.Z]
END_VISUALIZATION

// ---- VISUs/visu_ReM.TcVIS
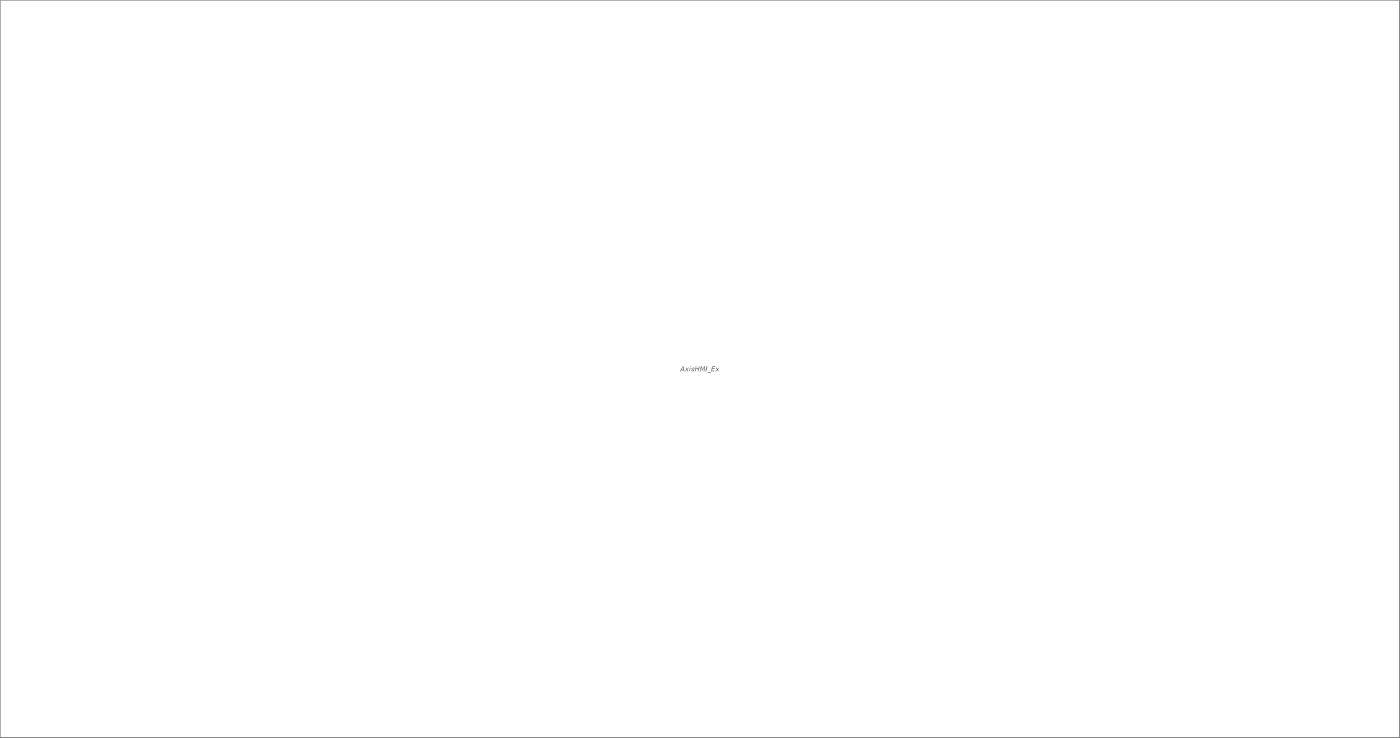
VISUALIZATION visu_ReM  // 2048x1080
    TabControl (0,0 2048x1080)
        shows AxisHMI_Ex(stAxisHMI := GVL.rem[G_HMI.iReM].lift[0].st_mcAxis, mcAxis := GVL.rem[G_HMI.iReM].lift[0].mcAxis, xError := GVL.rem[G_HMI.iReM].lift[0].mcAxis.xError)
        shows AxisHMI_Ex(stAxisHMI := GVL.rem[G_HMI.iReM].lift[1].st_mcAxis, mcAxis := GVL.rem[G_HMI.iReM].lift[1].mcAxis, xError := GVL.rem[G_HMI.iReM].lift[1].mcAxis.xError)
        shows v_rem_0(dIO_ReM := GVL.rem[G_HMI.iReM])
        shows v_rem_1(dIO_ReM := GVL.rem[G_HMI.iReM])
        shows Axis_HMI(st_axis_HMI := st_mcAxis[EN_Axis.Grip_axis])
        [0]: TabTitle=Lift0
        [1]: TabTitle=Lift1
        [2]: TabTitle=ReMIO_0, AxisHMI=gantrybase.st_mcAxis[EN_Axis.Z], mcAxis=gantrybase.mcAxis[EN_Axis.Z], Error=gantrybase.mcAxis[EN_Axis.Z].xError
        [3]: TabTitle=ReMIO_1
        [6]: TabTitle=Gripper
        p699000190: gantrybase.st_mcAxis[EN_Axis.X]
        p2837713833: gantrybase.mcAxis[EN_Axis.Z].sAxisName
        p520277221: gantrybase.mcAxis[EN_Axis.X].xError
        p3331604638: gantrybase.st_mcAxis[EN_Axis.Z]
        p1813558639: gantrybase.mcAxis[EN_Axis.Z].xError
        p1563495665: gantrybase.st_mcAxis[EN_Axis.Y]
        p2070126892: gantrybase.mcAxis[EN_Axis.Y].xError
        p3435970784: gantrybase.mcAxis[EN_Axis.X]
        p2829954345: gantrybase.mcAxis[EN_Axis.Y]
        p3218520426: gantrybase.mcAxis[EN_Axis.Z]
END_VISUALIZATION

// ---- VISUs/visu_MLC.TcVIS
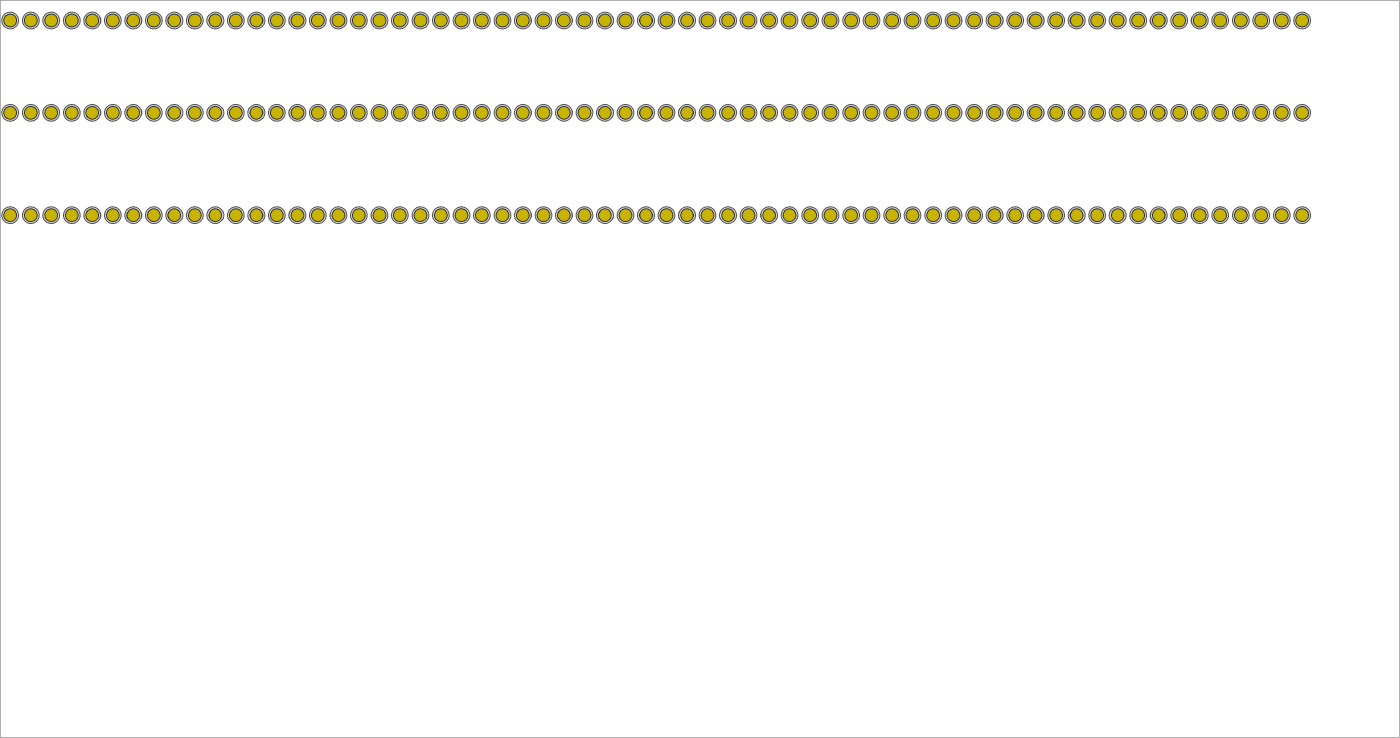
VISUALIZATION visu_MLC  // 2048x1080
    Frame (0,15 240x30)
        shows v_byte(iNum := GVL.ibyteNum[1])
    Frame (0,300 240x30)
        shows v_byte(iNum := GVL.ibyteNum[17])
    Frame (240,300 240x30)
        shows v_byte(iNum := GVL.ibyteNum[18])
    Frame (480,300 240x30)
        shows v_byte(iNum := GVL.ibyteNum[19])
    Frame (720,300 240x30)
        shows v_byte(iNum := GVL.ibyteNum[20])
    Frame (960,300 240x30)
        shows v_byte(iNum := GVL.ibyteNum[21])
    Frame (1200,300 240x30)
        shows v_byte(iNum := GVL.ibyteNum[22])
    Frame (1440,300 240x30)
        shows v_byte(iNum := GVL.ibyteNum[23])
    Frame (1680,300 240x30)
        shows v_byte(iNum := GVL.ibyteNum[24])
    Frame (0,150 240x30)
        shows v_byte(iNum := GVL.ibyteNum[9])
    Frame (240,150 240x30)
        shows v_byte(iNum := GVL.ibyteNum[10])
    Frame (480,150 240x30)
        shows v_byte(iNum := GVL.ibyteNum[11])
    Frame (720,150 240x30)
        shows v_byte(iNum := GVL.ibyteNum[12])
    Frame (960,150 240x30)
        shows v_byte(iNum := GVL.ibyteNum[13])
    Frame (1200,150 240x30)
        shows v_byte(iNum := GVL.ibyteNum[14])
    Frame (1440,150 240x30)
        shows v_byte(iNum := GVL.ibyteNum[15])
    Frame (1680,150 240x30)
        shows v_byte(iNum := GVL.ibyteNum[16])
    Frame (240,15 240x30)
        shows v_byte(iNum := GVL.ibyteNum[2])
    Frame (480,15 240x30)
        shows v_byte(iNum := GVL.ibyteNum[3])
    Frame (720,15 240x30)
        shows v_byte(iNum := GVL.ibyteNum[4])
    Frame (960,15 240x30)
        shows v_byte(iNum := GVL.ibyteNum[5])
    Frame (1200,15 240x30)
        shows v_byte(iNum := GVL.ibyteNum[6])
    Frame (1440,15 240x30)
        shows v_byte(iNum := GVL.ibyteNum[7])
    Frame (1680,15 240x30)
        shows v_byte(iNum := GVL.ibyteNum[8])
END_VISUALIZATION

// ---- VISUs/visu_main.TcVIS
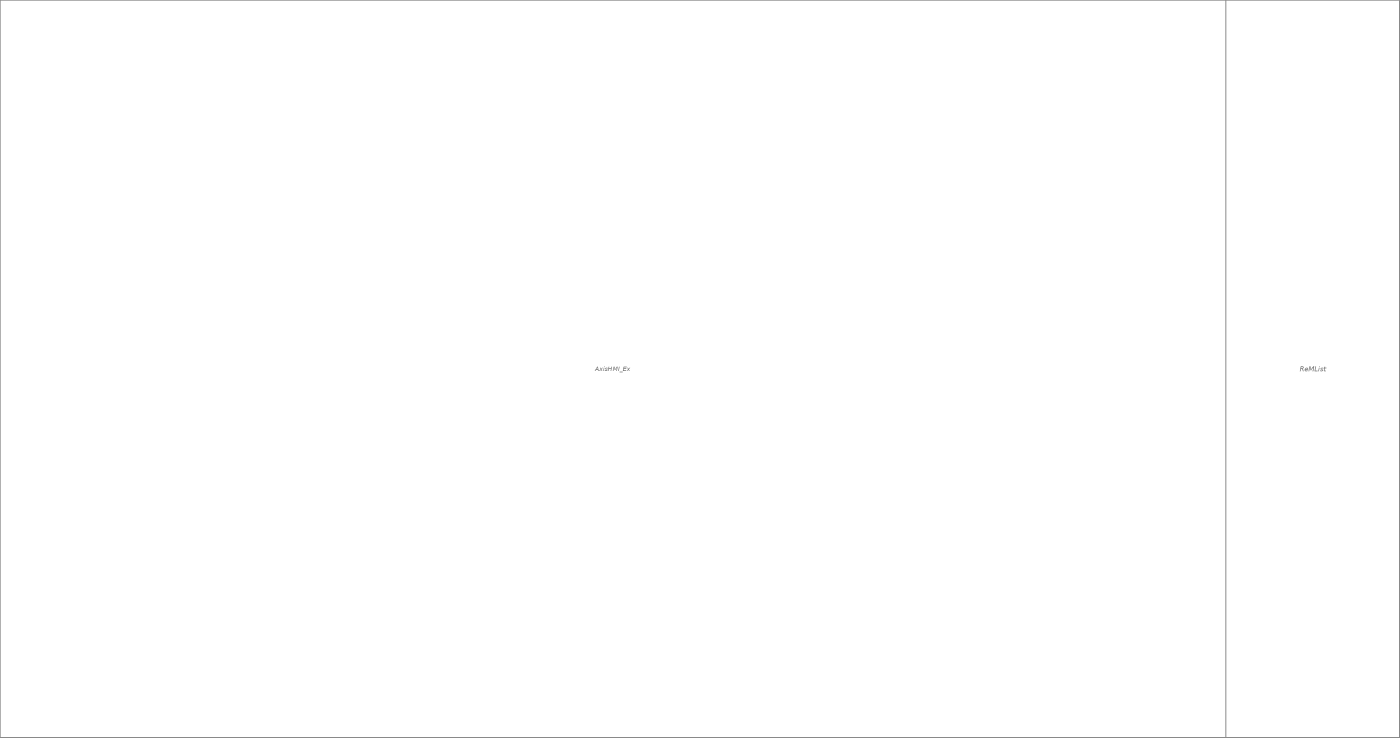
VISUALIZATION visu_main  // 2048x1080
    TabControl (1793,0 255x1080)
        shows ReMList()
        shows PMList()
        shows OtherList()
        shows Visualization_4()
        [0]: TabTitle=ReM
        [2]: TabTitle=Others
    Frame (0,0 1793x1080), frame switch variable: G_HMI.iMainFrame
        shows visu_ReM()
        shows visu_PM()
END_VISUALIZATION

// ---- VISUs/ReMList.TcVIS
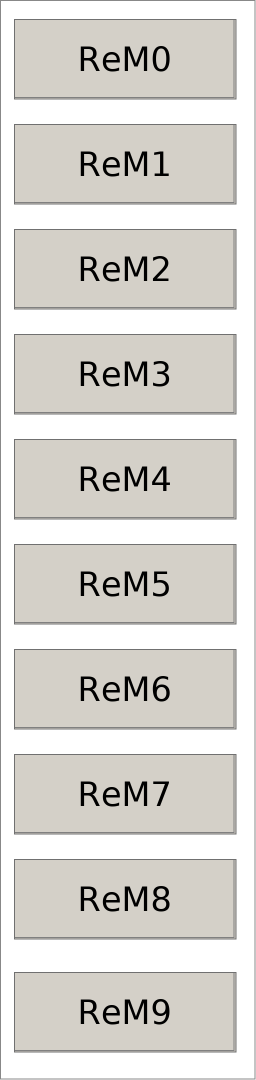
VISUALIZATION ReMList  // 256x1080
    Button (14,19 222x80), "ReM0", colour toggle: G_HMI.iReM =0
        p573394764: 16#FF00FF00
        OnMouseDown: execute { G_HMI.iReM  := 0; G_HMI.iMainFrame	:= 0; }
    Button (14,124 222x80), "ReM1", colour toggle: G_HMI.iReM =1
        p573394764: 16#FF00FF00
        OnMouseDown: execute { G_HMI.iReM  := 1; G_HMI.iMainFrame	:= 0; }
    Button (14,229 222x80), "ReM2", colour toggle: G_HMI.iReM =2
        p573394764: 16#FF00FF00
        OnMouseDown: execute { G_HMI.iReM  := 2; G_HMI.iMainFrame	:= 0; }
    Button (14,334 222x80), "ReM3", colour toggle: G_HMI.iReM =3
        p573394764: 16#FF00FF00
        OnMouseDown: execute { G_HMI.iReM  := 3; G_HMI.iMainFrame	:= 0; }
    Button (14,439 222x80), "ReM4", colour toggle: G_HMI.iReM =4
        p573394764: 16#FF00FF00
        OnMouseDown: execute { G_HMI.iReM  := 4; G_HMI.iMainFrame	:= 0; }
    Button (14,544 222x80), "ReM5", colour toggle: G_HMI.iReM =5
        p573394764: 16#FF00FF00
        OnMouseDown: execute { G_HMI.iReM  := 5; G_HMI.iMainFrame	:= 0; }
    Button (14,649 222x80), "ReM6", colour toggle: G_HMI.iReM =6
        p573394764: 16#FF00FF00
        OnMouseDown: execute { G_HMI.iReM  := 6; G_HMI.iMainFrame	:= 0; }
    Button (14,754 222x80), "ReM7", colour toggle: G_HMI.iReM =7
        p573394764: 16#FF00FF00
        OnMouseDown: execute { G_HMI.iReM  := 7; G_HMI.iMainFrame	:= 0; }
    Button (14,859 222x80), "ReM8", colour toggle: G_HMI.iReM =8
        p573394764: 16#FF00FF00
        OnMouseDown: execute { G_HMI.iReM  := 8; G_HMI.iMainFrame	:= 0; }
    Button (14,972 222x80), "ReM9", colour toggle: G_HMI.iReM =9
        p573394764: 16#FF00FF00
        OnMouseDown: execute { G_HMI.iReM  := 9; G_HMI.iMainFrame	:= 0; }
END_VISUALIZATION

// ---- VISUs/PMList.TcVIS
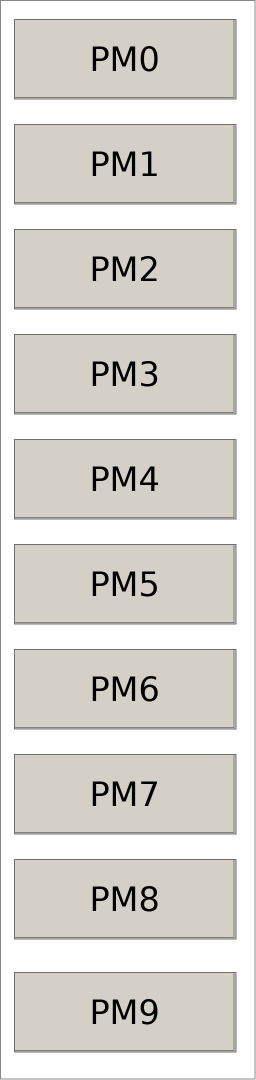
VISUALIZATION PMList  // 256x1080
    Button (1413,1160 244x110), "ReM0"
        OnMouseDown: execute { G_HMI.iMainFrame  := 0; }
    Button (14,19 222x80), "PM0", colour toggle: G_HMI.iPM =0
        p573394764: 16#FF00FF00
        OnMouseDown: execute { G_HMI.iPM  := 0; G_HMI.iMainFrame	:= 1; }
    Button (14,124 222x80), "PM1", colour toggle: G_HMI.iPM =1
        p573394764: 16#FF00FF00
        OnMouseDown: execute { G_HMI.iPM  := 1; G_HMI.iMainFrame	:= 1; }
    Button (14,229 222x80), "PM2", colour toggle: G_HMI.iPM =2
        p573394764: 16#FF00FF00
        OnMouseDown: execute { G_HMI.iPM  := 2; G_HMI.iMainFrame	:= 1; }
    Button (14,334 222x80), "PM3", colour toggle: G_HMI.iPM =3
        p573394764: 16#FF00FF00
        OnMouseDown: execute { G_HMI.iPM  := 3; G_HMI.iMainFrame	:= 1; }
    Button (14,439 222x80), "PM4", colour toggle: G_HMI.iPM =4
        p573394764: 16#FF00FF00
        OnMouseDown: execute { G_HMI.iPM  := 4; G_HMI.iMainFrame	:= 1; }
    Button (14,544 222x80), "PM5", colour toggle: G_HMI.iPM =5
        p573394764: 16#FF00FF00
        OnMouseDown: execute { G_HMI.iPM  := 5; G_HMI.iMainFrame	:= 1; }
    Button (14,649 222x80), "PM6", colour toggle: G_HMI.iReM =6
        p573394764: 16#FF00FF00
        OnMouseDown: execute { G_HMI.iPM  := 6; G_HMI.iMainFrame	:= 1; }
    Button (14,754 222x80), "PM7", colour toggle: G_HMI.iReM =7
        p573394764: 16#FF00FF00
        OnMouseDown: execute { G_HMI.iPM  := 7; G_HMI.iMainFrame	:= 1; }
    Button (14,859 222x80), "PM8", colour toggle: G_HMI.iReM =8
        p573394764: 16#FF00FF00
        OnMouseDown: execute { G_HMI.iPM  := 8; G_HMI.iMainFrame	:= 1; }
    Button (14,972 222x80), "PM9", colour toggle: G_HMI.iReM =9
        p573394764: 16#FF00FF00
        OnMouseDown: execute { G_HMI.iPM  := 9; G_HMI.iMainFrame	:= 1; }
END_VISUALIZATION

